(* CODESYS project RepoTestGitCodesys2

Project tree, tasks and I/O mapping:
  Device : CODESYS Control Win V3, 3S - Smart Software Solutions GmbH, version 3.5.19.50
    application Application
      libraries: Standard, 3.5.18.0 (System); Util, 3.5.19.0 (System); Building Automation, 1.0.0.0 (CODESYS Group); CmpBitmapPool, * (System); BASIC, 3.31 (OSCAT); SysTime, 3.5.17.0 (System); SysTypes Interfaces, * (System)
      task AlarmManagerTask (cyclic, interval 50 ms, priority 31) calls AlarmManager.Alarm_Prg
      task MainTask (cyclic, interval t#20ms, priority 1) calls PLC_PRG, test_CFC
      task VISU_TASK (cyclic, interval 100 ms, priority 31) calls VisuElems.Visu_Prg
      Alarm Configuration
        alarm class Alarm (priority 0, acknowledge ACK)
        AlarmStorage
        alarm class Error (priority 10, acknowledge REP)
        alarm class Info (priority 100, acknowledge REP)
        text list List_alarm
        alarm group List_alarm
            0 [Alarm]: Comparison Equal, ExpressionToCompare TRUE, Expression (Reaktor1.Pause.PP00_LT01.WH OR Reaktor1.Innpumping.PP00_LT01.WH) - "Høgt nivå mottakstankl"
            1 [Alarm]: Comparison Equal, ExpressionToCompare TRUE, Expression (Reaktor1.Pause.PP00_LT01.WL OR Reaktor1.Innpumping.PP00_LT01.WL) - "Lavt nivå mottakstank"
            10 [Alarm]: Comparison Equal, ExpressionToCompare TRUE, Expression ((Reaktor2.Pause.PP02_LT02.WL OR Reaktor2.Innpumping.PP02_LT02.WL) OR Reaktor2.Uttaping.PP02_LT02.WL)
            11 [Alarm]: Comparison Equal, ExpressionToCompare TRUE, Expression GVL_Inputs.IA01_PR01_WH
            12 [Alarm]: Comparison Equal, ExpressionToCompare TRUE, Expression GVL_Inputs.IA01_PR01_WL
            13 [Alarm]: Comparison Equal, ExpressionToCompare TRUE, Expression GVL_Inputs.Water_sensor
            2 [Alarm]: Comparison Equal, ExpressionToCompare TRUE, Expression GVL_Inputs.WH_Overflow - "Anlegg i overløp"
            3 [Alarm]: Comparison Equal, ExpressionToCompare TRUE, Expression GVL_Inputs.PA01_PR01_WH
            4 [Alarm]: Comparison Equal, ExpressionToCompare TRUE, Expression GVL_Inputs.PA01_PR01_WL
            5 [Alarm]: Comparison Equal, ExpressionToCompare TRUE, Expression GVL_Inputs.PA02_PR01_WH
            6 [Alarm]: Comparison Equal, ExpressionToCompare TRUE, Expression GVL_Inputs.PA02_PR01_WL
            7 [Alarm]: Comparison Equal, ExpressionToCompare TRUE, Expression ((Reaktor1.Pause.PP01_LT01.WH OR Reaktor1.Innpumping.PP01_LT01.WH) OR Reaktor1.Uttaping.PP01_LT01.WH)
            8 [Alarm]: Comparison Equal, ExpressionToCompare TRUE, Expression ((Reaktor1.Pause.PP01_LT01.WL OR Reaktor1.Innpumping.PP01_LT01.WL) OR Reaktor1.Uttaping.PP01_LT01.WL)
            9 [Alarm]: Comparison Equal, ExpressionToCompare TRUE, Expression ((Reaktor2.Pause.PP02_LT02.WH OR Reaktor2.Innpumping.PP02_LT02.WH) OR Reaktor2.Uttaping.PP02_LT02.WH)
        text list List_Error
        alarm group List_Error
            0 [Error]: Comparison Equal, ExpressionToCompare TRUE, Expression GVL_Inputs.XF_Huber - "Feilsignal grovrist"
            1 [Error]: Comparison Equal, ExpressionToCompare TRUE, Expression Reaktor1.Pause.PP00_LT01.YF OR Reaktor1.Innpumping.PP00_LT01.YF - "Feil på trykkgivar mottakstank"
            10 [Error]: Comparison Equal, ExpressionToCompare TRUE, Expression ((Reaktor1.Innpumping.PP01_PS01.YF = TRUE) AND (Reaktor1.Innpumping.PP01_PS01.YFI = 6)) - "Feil matepumpe 1, safeguard blocking konflikt"
            11 [Error]: Comparison Equal, ExpressionToCompare TRUE, Expression ((Reaktor1.Innpumping.PP01_PS01.YF = TRUE) AND (Reaktor1.Innpumping.PP01_PS01.YFI = 7)) - "Feil matepumpe 1, safeguard mangel tilbakemelding"
            12 [Error]: Comparison Equal, ExpressionToCompare TRUE, Expression ((Reaktor1.Innpumping.PP01_PS01.YF = TRUE) AND (Reaktor1.Innpumping.PP01_PS01.YFI = 8)) - "Feil matepumpe 1, tap av aktivering"
            13 [Error]: Comparison Equal, ExpressionToCompare TRUE, Expression GVL_Inputs.PP01_PS01_XF - "Motorvern matepumpe 1 utløyst"
            14 [Error]: Comparison Equal, ExpressionToCompare TRUE, Expression ((Reaktor1.Innpumping.PP02_PS01.YF = TRUE) AND (Reaktor1.Innpumping.PP02_PS01.YFI = 1)) - "Feil matepumpe 2, mista tilbakemelding høg"
            15 [Error]: Comparison Equal, ExpressionToCompare TRUE, Expression ((Reaktor1.Innpumping.PP02_PS01.YF = TRUE) AND (Reaktor1.Innpumping.PP02_PS01.YFI = 2))
            16 [Error]: Comparison Equal, ExpressionToCompare TRUE, Expression ((Reaktor1.Innpumping.PP02_PS01.YF = TRUE) AND (Reaktor1.Innpumping.PP02_PS01.YFI = 3))
            17 [Error]: Comparison Equal, ExpressionToCompare TRUE, Expression ((Reaktor1.Innpumping.PP02_PS01.YF = TRUE) AND (Reaktor1.Innpumping.PP02_PS01.YFI = 4))
            18 [Error]: Comparison Equal, ExpressionToCompare TRUE, Expression ((Reaktor1.Innpumping.PP02_PS01.YF = TRUE) AND (Reaktor1.Innpumping.PP02_PS01.YFI = 5))
            19 [Error]: Comparison Equal, ExpressionToCompare TRUE, Expression ((Reaktor1.Innpumping.PP02_PS01.YF = TRUE) AND (Reaktor1.Innpumping.PP02_PS01.YFI = 6))
            2 [Error]: Comparison Equal, ExpressionToCompare TRUE, Expression Reaktor1.Pause.PP00_LS01.YF OR Reaktor1.Innpumping.PP00_LS01.YF - "Feil på nivåvippe lav mottakstank"
            20 [Error]: Comparison Equal, ExpressionToCompare TRUE, Expression ((Reaktor1.Innpumping.PP02_PS01.YF = TRUE) AND (Reaktor1.Innpumping.PP02_PS01.YFI = 7))
            21 [Error]: Comparison Equal, ExpressionToCompare TRUE, Expression ((Reaktor1.Innpumping.PP02_PS01.YF = TRUE) AND (Reaktor1.Innpumping.PP02_PS01.YFI = 8))
            22 [Error]: Comparison Equal, ExpressionToCompare TRUE, Expression GVL_Inputs.PP02_PS01_XF
            23 [Error]: Comparison Equal, ExpressionToCompare TRUE, Expression ((Reaktor1.Innpumping.PP01_VP01.YF = TRUE) AND (Reaktor1.Innpumping.PP01_VP01.YF = 1))
            24 [Error]: Comparison Equal, ExpressionToCompare TRUE, Expression ((Reaktor1.Innpumping.PP01_VP01.YF = TRUE) AND (Reaktor1.Innpumping.PP01_VP01.YF = 2))
            25 [Error]: Comparison Equal, ExpressionToCompare TRUE, Expression ((Reaktor1.Innpumping.PP01_VP01.YF = TRUE) AND (Reaktor1.Innpumping.PP01_VP01.YF = 3))
            26 [Error]: Comparison Equal, ExpressionToCompare TRUE, Expression ((Reaktor1.Innpumping.PP01_VP01.YF = TRUE) AND (Reaktor1.Innpumping.PP01_VP01.YF = 4))
            27 [Error]: Comparison Equal, ExpressionToCompare TRUE, Expression ((Reaktor1.Innpumping.PP01_VP01.YF = TRUE) AND (Reaktor1.Innpumping.PP01_VP01.YF = 5))
            28 [Error]: Comparison Equal, ExpressionToCompare TRUE, Expression ((Reaktor1.Innpumping.PP01_VP01.YF = TRUE) AND (Reaktor1.Innpumping.PP01_VP01.YF = 6))
            29 [Error]: Comparison Equal, ExpressionToCompare TRUE, Expression ((Reaktor1.Innpumping.PP01_VP01.YF = TRUE) AND (Reaktor1.Innpumping.PP01_VP01.YF = 7))
            3 [Error]: Comparison Equal, ExpressionToCompare TRUE, Expression (Reaktor1.Pause.PP00_LS02.YF OR Reaktor1.Innpumping.PP00_LS02.YF) - "Feil på nivåvippe høg mottakstank"
            4 [Error]: Comparison Equal, ExpressionToCompare TRUE, Expression GVL_Inputs.XF_Overflow - "Feil på trykkgivar overløp"
            5 [Error]: Comparison Equal, ExpressionToCompare TRUE, Expression ((Reaktor1.Innpumping.PP01_PS01.YF = TRUE) AND (Reaktor1.Innpumping.PP01_PS01.YFI = 1)) - "Feil matepumpe 1, mista tilbakemeldig høg"
            6 [Error]: Comparison Equal, ExpressionToCompare TRUE, Expression ((Reaktor1.Innpumping.PP01_PS01.YF = TRUE) AND (Reaktor1.Innpumping.PP01_PS01.YFI = 2)) - "Feil matepumpe 1, mista tilbakemelding lav"
            7 [Error]: Comparison Equal, ExpressionToCompare TRUE, Expression ((Reaktor1.Innpumping.PP01_PS01.YF = TRUE) AND (Reaktor1.Innpumping.PP01_PS01.YFI = 3)) - "Feil matepumpe 1, mangel tilbakemelding høg"
            8 [Error]: Comparison Equal, ExpressionToCompare TRUE, Expression ((Reaktor1.Innpumping.PP01_PS01.YF = TRUE) AND (Reaktor1.Innpumping.PP01_PS01.YFI = 4)) - "Feil matepumpe 1, mangel tilbakemelding lav"
            9 [Error]: Comparison Equal, ExpressionToCompare TRUE, Expression ((Reaktor1.Innpumping.PP01_PS01.YF = TRUE) AND (Reaktor1.Innpumping.PP01_PS01.YFI = 5)) - "Feil matepumpe 1, ekstern feil"
        alarm group List_Info
        text list List_Info
        alarm group List_Warning
        text list List_Warning
        alarm class Warning (priority 30, acknowledge REP)
      function block BUGS [ST]
      Common_Functions/
        program CommonFunctions [CFC]
        function block Pumphouse [CFC]
      function block fbAnalougeAlarm [ST]
      function block fbDigitalAlarm [ST]
      function block fbInnpumping [ST]
      function block fbPause [ST]
      function block fbSwap [ST]
      function block fbTimer [ST]
      function block fbUtrekningar [ST]
      Function blocks/
        function block Fault_Mapping [ST]
        function block fbBehandlaVatn [ST]
        function block fbCAC [ST]
        function block fbDatabehandling [ST]
        function block fbFeilhandtering [ST]
        function block fbHighload [ST]
        function block fbPumphouse [ST]
        function block fbPumpInterlock [ST]
        function block fbReaksjon [ST]
        function block fbSedementering [ST]
        function block fbSivbedRotation [ST]
        function block fbSlamutak [ST]
        function block fbUttapping [ST]
        function block Output_Mapping [ST]
      Function blocks/
      Functions/
        function Volume_Rectangle [ST]
      Global Variable Lists/
        global variables GVL_Outputs
        global variables GVL_Rest
      global variables GVL
      global variables GVL_Inputs
      global variables GVL_R1
      global variables GVL_R2
      global variables GVL_Sekvenstider
      global variables GVL_TM
      Heile_R1/
        function block R1_Innpumping [CFC]
        function block R1_Pause [CFC]
        function block R1_Reaksjon [CFC]
        function block R1_Sedementering [CFC]
        function block R1_Slam [CFC]
        function block R1_Uttapping [CFC]
        program Reaktor1 [CFC]
      Heile_R2/
        function block R2_Innpumping [CFC]
        function block R2_Innpumping [CFC]
        function block R2_Pause [CFC]
        function block R2_Pause [CFC]
        function block R2_Reaksjon [CFC]
        function block R2_Sedementering [CFC]
        function block R2_Slam [CFC]
        function block R2_Uttapping [CFC]
        program Reaktor2 [CFC]
        program Reaktor2 [CFC]
      function IEC_Time [ST]
      image pool ImagePool
      function block MA [ST]
      function block MB [ST]
      text list MyStates
      program PLC_PRG [ST]
      program POU [ST]
      function block SBE [ST]
      function block SBV [ST]
      function block SBV [ST]
      function block SBV_ReArranged [ST]
      Simulation/
        function block Analog_I [LD]
        function block Analog_O [LD]
        function block fbTankTest [ST]
        function block fbTankVirk [LD]
        function block fbValveSim [ST]
        function block ManualControl [LD]
        global variables Simu
        program Simulering [CFC]
        program Tank [ST]
      visualisation Simulering
      function block SPE [ST]
      visualisation Symbol
      Test_Blocks/
        function block SBV_1 [ST]
        function block test [ST]
        program Reaktor_2 [CFC]
      program test_CFC [CFC]
      function block test [CFC]
      program test_SFC [SFC]: Init_active
      visualisation Testing
      Tilstandsmaskin/
      function block tmReactor1 [ST]
      program Utrekningar [ST]
      function VolumReaktor [ST]
  libraries: VisuSymbols, 4.5.0.0 (System)
  5ce3da45-db07-42e7-a21c-a00fff4ed8f6|C:\Users\Peter\Downloads\GreenBlaser.png
  5ce3da45-db07-42e7-a21c-a00fff4ed8f6|C:\Users\Peter\Downloads\GreenPump90d.png
  5ce3da45-db07-42e7-a21c-a00fff4ed8f6|C:\Users\Peter\Downloads\GreenPump.png
  5ce3da45-db07-42e7-a21c-a00fff4ed8f6|C:\Users\Peter\Downloads\GreenValve-removebg-preview.png
  5ce3da45-db07-42e7-a21c-a00fff4ed8f6|C:\Users\Peter\Downloads\SARA (2).png
  5ce3da45-db07-42e7-a21c-a00fff4ed8f6|C:\Users\Peter\Downloads\WhiteBlaser.png
  5ce3da45-db07-42e7-a21c-a00fff4ed8f6|C:\Users\Peter\Downloads\WhitePump90d.png
  5ce3da45-db07-42e7-a21c-a00fff4ed8f6|C:\Users\Peter\Downloads\WhitePump.png
  5ce3da45-db07-42e7-a21c-a00fff4ed8f6|C:\Users\Peter\Downloads\WhiteValve-removebg-preview.png
  5ce3da45-db07-42e7-a21c-a00fff4ed8f6|C:\Users\Peter\OneDrive - Høgskulen på Vestlandet\Mango_Disk\Bachelor RA200 Sande\Dokumentasjon\P&ID\Eldre versjoner\SARA_P&ID_rev2.drawio.png
  5ce3da45-db07-42e7-a21c-a00fff4ed8f6|C:\Users\Peter\OneDrive - Høgskulen på Vestlandet\Mango_Disk\Bachelor RA200 Sande\Dokumentasjon\P&ID\P&ID Automatisk styrt.png
  5ce3da45-db07-42e7-a21c-a00fff4ed8f6|C:\Users\Peter\OneDrive - Renasys\Dokumenter\GreenValve90d.png
  5ce3da45-db07-42e7-a21c-a00fff4ed8f6|C:\Users\Peter\OneDrive - Renasys\Dokumenter\WhiteValve90d.png
  5ce3da45-db07-42e7-a21c-a00fff4ed8f6|C:\Users\Peter\OneDrive - Renasys\Skrivebord\GreenValve.png
  5ce3da45-db07-42e7-a21c-a00fff4ed8f6|C:\Users\Peter\OneDrive - Renasys\Skrivebord\WhiteValve.png
  5ce3da45-db07-42e7-a21c-a00fff4ed8f6|C:\Users\Peter\OneDrive\Skrivebord\test.png
  GlobalImagePool
  text list GlobalTextList
*)

// Device/Application/GVL
{attribute 'qualified_only'}


VAR_GLOBAL
	lvlTransmitter_Mottak : REAL;
	
END_VAR

// Device/Application/GVL_Inputs
{attribute 'qualified_only'}
VAR_GLOBAL
	
END_VAR

// Device/Application/GVL_R1
{attribute 'qualified_only'}
VAR_GLOBAL
	// Reaktor 1 INPUT	
	SekvensPauseOK					: BOOL;		// Sekvense Pause 			gjennomført
	SekvensInnpumpingOK				: BOOL;		// Sekvense Innpumping  	gjennomført
	SekvensReaksjonOK				: BOOL;		// Sekvense Reaksjon 		gjennomført
	SekvensSedimenteringOK			: BOOL;		// Sekvense Sedimentering 	gjennomført
	SekvensUttappingOK				: BOOL;		// Sekvense Uttapping 		gjennomført

	// Reaktor 1 OUTPUT
	Pause							: BOOL;		// [TRUE] Aktiv Sekvens Pause
	Innpumping 						: BOOL;		// [TRUE] Aktiv Sekvens Innpumping
	Reaksjon 						: BOOL;		// [TRUE] Aktiv Sekvens Reaksjon
	Sedimentering 					: BOOL;		// [TRUE] Aktiv Sekvens Sedimentering
	Uttapping						: BOOL;		// [TRUE] Aktiv Sekvens Uttapping
	
	// Reaktor 1 Sekvens Tider	
	SekvenstidInnpumping			: TIME;		// Maks tid innpumpingssekvens
	SekvenstidReaksjon				: TIME;		// Maks tid reaksjonssekvens
	SekvenstidSedimentering			: TIME;		// Maks tid sedimenteringssekvens
	SekvenstidUttapping  			: TIME;		// Maks tid Uttapping
	
	// Reaktor 1 Reaksjonstider
	GangtidAnoks					: TIME;		// Gangtid Anoks reaksjonsfase 
	GangtidAerob					: TIME;		// Gangtid Aerob reaksjonsfase
	GangtidKjemikalieDosering		: TIME;		// Gangtid Kjemikaliepumpe
	SikkerheitsIntervallKjemikalie	: TIME;		// Tid mellom ferdig kjemikaliedosering og slutt reaksjonsfase : SekvenstidReaksjon - (GangtidKjemikalieDosering + SikkerheitsIntervallKjemikalie)
END_VAR

// Device/Application/GVL_R2
{attribute 'qualified_only'}
VAR_GLOBAL
	// Reaktor 2 INPUT	
	SekvensPauseOK					: BOOL;		// Sekvense Pause 			gjennomført
	SekvensInnpumpingOK				: BOOL;		// Sekvense Innpumping  	gjennomført
	SekvensReaksjonOK				: BOOL;		// Sekvense Reaksjon 		gjennomført
	SekvensSedimenteringOK			: BOOL;		// Sekvense Sedimentering 	gjennomført
	SekvensUttappingOK				: BOOL;		// Sekvense Uttapping 		gjennomført

	// Reaktor 2 OUTPUT
	Pause							: BOOL;		// [TRUE] Aktiv Sekvens Pause							
	Innpumping 						: BOOL;		// [TRUE] Aktiv Sekvens Innpumping
	Reaksjon 						: BOOL;		// [TRUE] Aktiv Sekvens Reaksjon
	Sedementering 					: BOOL;		// [TRUE] Aktiv Sekvens Sedimentering
	Uttapping						: BOOL;		// [TRUE] Aktiv Sekvens Uttapping
	
	// Reaktor 2 Sekvens Tider
	SekvenstidInnpumping			: TIME;		// Maks tid innpumpingssekvens
	SekvenstidReaksjon				: TIME;		// Maks tid reaksjonssekvens
	SekvenstidSedimentering			: TIME;		// Maks tid sedimenteringssekvens
	SekvenstidUttapping  			: TIME;		// Maks tid Uttapping
	
	// Reaktor 2 Reaksjonstider
	GangtidAnoks					: TIME;		// Gangtid Anoks reaksjonsfase
	GangtidAerob					: TIME;		// Gangtid Aerob reaksjonsfase
	GangtidKjemikalie				: TIME;		// Gangtid Kjemikaliepumpe
	SikkerheitsIntervallKjemikalie	: TIME;		// Tid mellom ferdig kjemikaliedosering og slutt reaksjonsfase : SekvenstidReaksjon - (GangtidKjemikalieDosering + SikkerheitsIntervallKjemikalie)
END_VAR

// Device/Application/GVL_Sekvenstider
{attribute 'qualified_only'}
VAR_GLOBAL	
	TidInnpumpingMaks			: TIME := T#10S;
	TidReaksjon					: TIME := T#3S;
	TidSedimentering			: TIME := T#3S;
	TidUttapping  				: TIME := T#3S;
END_VAR

// Device/Application/GVL_TM
{attribute 'qualified_only'}
VAR_GLOBAL
	
	// Reaktor 1
	Pause1						: BOOL;							//
	Innpumping1 				: BOOL;
	Innpumping_Pause1			: BOOL;
	Reaksjon1 					: BOOL;
	Sedementering1 				: BOOL;
	Uttapping1					: BOOL;
	
	// Reaktor 2
	Pause2						: BOOL;							//
	Innpumping2 				: BOOL;
	Innpumping_Pause2			: BOOL;
	Reaksjon2 					: BOOL;
	Sedementering2 				: BOOL;
	Uttapping2					: BOOL;
	
	// Til tilstandsmaskin
	PauseReaktor1OK				: BOOL;
	
	InnpumpingReaktor1OK		: BOOL; 
	InnpumpingReaktor1Pause		: BOOL;
END_VAR

// Device/Application/Global Variable Lists/GVL_Outputs
{attribute 'qualified_only'}
VAR_GLOBAL
END_VAR

// Device/Application/Global Variable Lists/GVL_Rest
{attribute 'qualified_only'}
VAR_GLOBAL
	
	MottakstankNivaa	: REAL;
	MottakstankVolum	: REAL;
	siSivState			: INT;
	GangerPrSivBed		: INT;

END_VAR

// Device/Application/Simulation/Simu
{attribute 'qualified_only'}
VAR_GLOBAL
	XE	: BOOL := TRUE;
	LA	: BOOL;
	
	MTankNivaa		: REAL;
	R1Nivaa			: REAL;
	FlowInlet		: INT;
	FlowOutletR1	: INT;
	
	PP01_VP01_YF 	: BOOL;
	PP02_VP01_YF 	: BOOL;
	TW02_VH01_YF 	: BOOL;
	
	PP01_PS01_YF 	: BOOL;
	PP02_PS01_YF 	: BOOL;
	PA01_BL01_YF 	: BOOL;
	CH00_PH01_YF 	: BOOL;
END_VAR

// Device/Application/PLC_PRG
PROGRAM PLC_PRG
VAR

LS_LOW   : MB;
LS_HIGH  : MB;
PT_Tank	 : MA;
PT_R1	 : MA;
PT_R2	 : MA;
M1		 : SPE;
M2		 : SPE;
Valve1   : SBV;
Valve2	 : SBV;
Swap	 : fbSwap;

END_VAR

//Test();

LS_LOW();
LS_HIGH();
PT_TANK();
M1();
M2();
Valve1();
Valve2();
test();

// Beginning of the code :

IF LS_LOW.X THEN
	
	// Retracting Low Commands
	M1.XL		:= FALSE;
	Valve1.XL	:= FALSE;

	// Sending High Commands
	M1.XH 		:= TRUE;
	Valve1.XH 	:= TRUE;
	
ELSIF (NOT LS_LOW.X) THEN
	
	// Retracting HIGH Commands
	M1.XH		:= FALSE;
	Valve1.XH	:= FALSE;

	// Sending LOW Commands
	M1.XL 		:= TRUE;
	Valve1.XL 	:= TRUE;
	
END_IF

END_PROGRAM

// Device/Application/Test_Blocks/test
FUNCTION_BLOCK test
VAR_INPUT
END_VAR
VAR_OUTPUT
END_VAR
VAR
END_VAR

END_FUNCTION_BLOCK

// Device/Application/test
FUNCTION_BLOCK test
VAR_INPUT
	XE						: BOOL;			// Input from state machine
END_VAR
VAR_OUTPUT
	Y						: BOOL;			// Output to state machine
END_VAR

VAR
	// INPUT BLOCKS
	PP00_LS02   			: MB;			// Mottasktank vippe lav, call "Monitor Binary" 
	PP00_LS01  				: MB;			// Mottasktank vippe høg, call "Monitor Binary" 
	PP00_LT01	 			: MA;			// Mottasktank nivåmålar, call "Monitor Analog"
	PP01_LT01	 			: MA;			// Reaktor 1 nivåmålar,   call "Monitor Analog"
	
	// OUTPUT BLOCKS
	PA01_BL01				: SBE;			// Reaktor 1 blåser,	 call "Switch Binary Electrical"
	PP01_PS01		 		: SBE;			// Matepumpe 1,			 call "Switch Binary Electrical"
	PP02_PS01		 		: SBE;			// Matepumpe 2,			 call "Switch Binary Electrical"
	PP01_VP01   			: SBV;			// Reaktor 1 inn ventil, call "Switch Binary Valve"
	
	// FUNCTION BLOCKS
	Sekvens_Innpumping		: fbInnpumping;	// Innpumping logic,         call "fbInnpumping"
	Sim						: fbValveSim;	// Feedback balve simulator, call "fbValveSim"
END_VAR

VAR_TEMP		
	// FUNCTION CONTROL PARAMETERS
	PYHR				: REAL := 100;		// (Mottasktank nivåmålar & Reaktor 1 nivåmålar) MA Parameter Y high range
	PYLR				: REAL := 0;		// (Mottasktank nivåmålar & Reaktor 1 nivåmålar) MA Parameter Y low range
	PP00_LT01_PAHH		: REAL := 32;		// (Mottasktank nivåmålar) 						 MA Parameter high high action
	PP00_LT01_PALL		: REAL := 5;		// (Mottasktank nivåmålar) 						 MA Parameter low low action
	PP01_LT01_PAHH		: REAL := 90;		// (Reaktor 1 nivåmålar)   						 MA Parameter low low action 
	END_VAR

// -------------------------------------------------------------------------------------------------------------------------------------------------IN BLOCKS----------------------------------------------------------------------------------------------------------------------------------------------------------------------------------------------------------
// Mottakstank vippe høg
// INPUTS
// OUTPUTS
PP00_LS01(X := GVL_Inputs.PP00_LS01_X); // MB
// Mottakstank vippe lav
// INPUTS
// OUTPUTS
PP00_LS02(X := GVL_Inputs.PP00_LS02_X); // MB
// Mottakstank Nivåmåling
// INPUTS
PP00_LT01(
    X := GVL_Inputs.PP00_LT01_X,
    PAHH := PP00_LT01_PAHH,
    PALL := PP00_LT01_PALL,
    PYHR := PYHR,
    PYLR := PYLR); // MA
// OUTPUTS
GVL_Rest.MottakstankNivaa := PP00_LT01.Y;
// Reaktor 1 Nivåmåling
// INPUTS
PP01_LT01(X := GVL_Inputs.PP01_LT01_X, PAHH := PP01_LT01_PAHH, PYHR := PYHR, PYLR := PYLR); // MA
// OUTPUTS
GVL_R1.Nivaa := PP01_LT01.Y;
// ------------------------------------------------------------------------------------------------------------------------------------------------- CODE ----------------------------------------------------------------------------------------------------------------------------------------------------------------------------------------------------------
Sekvens_Innpumping(
    AHH_SendingTank := PP00_LT01.AHH,
    ALL_SendingTank := PP00_LT01.ALL,
    HH_SendingTank := PP00_LS01.Y,
    LL_Sending_Tank := PP00_LS02.Y,
    AHH_ReceivingTank := PP01_LT01.AHH,
    ALL_ReceivingTank := PP01_LT01.ALL,
    XGH_RValve := PP01_VP01.BCH,
    XGL_RValve := PP01_VP01.BCL,
    XGL_Pump1 := PP01_PS01.BCL,
    XGL_Pump2 := PP02_PS01.BCL,
    XE := XE,
    PIT := GVL_R1.SekvenstidInnpumping,
    PTI := GVL_R1.IntervallBlaser,
    PTD := GVL_R1.GangtidBlaser); // fbInnpumping
// Reaktor 1 blåser
// INPUTS
PA01_BL01(
    XGH := PA01_BL01.Y,
    XH := Sekvens_Innpumping.YH_Blower,
    XL := Sekvens_Innpumping.YL_Blower,
    XE := GVL_R1.Innpumping,
    LA := Simu.LA); // SBE
GVL_R1.Innpumping_PA01_BL01_YF := PA01_BL01.YF;
Y := Sekvens_Innpumping.Y;
// ------------------------------------------------------------------------------------------------------------------------------------------------- OUT BLOCKS  ---------------------------------------------------------------------------------------------------------------------------------------------------------------------------------------------------
// Inntaktspumpe 1
// INPUTS
PP01_PS01(
    XGH := PP01_PS01.Y,
    XH := Sekvens_Innpumping.YH_Pump1,
    XL := Sekvens_Innpumping.YL_Pump1,
    XE := GVL_R1.Innpumping,
    LA := Simu.LA); // SBE
GVL_R1.PP01_PS01_YF := PP01_PS01.YF;
// OUTPUTS
GVL_R1.PP01_PS01_Y := PP01_PS01.Y;
// Inntaktspumpe 2
// INPUTS
PP02_PS01(
    XGH := PP02_PS01.Y,
    XH := Sekvens_Innpumping.YH_Pump2,
    XL := Sekvens_Innpumping.YL_Pump2,
    XE := GVL_R1.Innpumping,
    LA := Simu.LA); // SBE
// OUTPUTS
GVL_R1.PP02_PS01_Y := PP02_PS01.Y;
GVL_R1.PP02_PS01_YF := PP02_PS01.YF;
// OUTPUTS
GVL_R1.Innpumping_PA01_BL01 := PA01_BL01.Y;
// Reaktor 1 inn ventil
// INPUTS
PP01_VP01(
    XGH := PP01_VP01.BCH,
    XGL := PP01_VP01.BCL,
    XH := Sekvens_Innpumping.YH_RValve,
    XL := Sekvens_Innpumping.YL_RValve,
    LA := Simu.LA); // SBV
// OUTPUTS
GVL_Outputs.PP01_VP01_Y := PP01_VP01.Y;
GVL_R1.PP01_VP01_YF := PP01_VP01.YF;
GVL_R1.PP01_VP01_BCH := PP01_VP01.BCH;

END_FUNCTION_BLOCK

// Device/Application/SBE
FUNCTION_BLOCK SBE
//The SBE function template shall be used for binary (on/off) control of flow element of medium 
//(electricity, heat or fluid). The controlled element is a unit, e.g. motor, pump, heater, fan etc.

VAR_INPUT
	{Signal FROM MCC, running status high (XGH = 1 is motor 
running)}
	XGH 		: BOOL; // Pos high feedback (MCC)	
	{XH = 1 (positive edge) set Y TO 1 in auto mode.)}
	XH 			: BOOL; // External set high 
	{XL = 1 (positive edge) set Y TO 0 in auto mode. XL is 
dominant over XH.}
	XL			: BOOL; // External set low
	{XOH = 1 set Y TO 1 in outside mode.}
	XOH 		: BOOL; // External outside set high
	{XOL = 1 set Y TO 0 in outside mode.}
	XOL			: BOOL; //External outside set low
	{Loop failure, e.g. I/O card broken}
	XF			: BOOL; // External fault
	{XE = 1 is required FOR a start. The effect on Y when XE goes 
low while running will be defined by parameter.}
	XE			: BOOL; // External enabled (MCC)
	{Safeguarding – LSH = 1. Overrule operator possibility TO 
operate Start/Stop and Auto/Manual. Locks template in 
manual mode and Y to 1 regardless of failure state. Input is 
subject to blocking. When signal goes low, the template 
remains in manual mode and Y = 1}
	LSH			: BOOL; // Lock safeguarding high
	{Safeguarding – LSL = 1 Overrule operator possibility TO 
operate Start/Stop and Auto/Manual. Locks template to 
manual mode and Y to 0 regardless of failure state. Input is 
subject to blocking. When signal goes low, the template 
remains in manual mode and Y = 0}
	LSL			: BOOL; // Lock safeguarding low
	{Safeguarding – FSH = 1 Overrule operator possibility TO 
operate Start/Stop. Sets Y to1 regardless of failure state. 
When signal is reset, the template will react to actual 
terminal statuses again. Signal is subject to blocking. If in 
Manual mode, the output (Y) remains 1 after signal returns 
to normal. }
	FSH			: BOOL; // Force safeguarding high
	{Safeguarding FSH = 0 Overrule operator possibility TO 
operate Start/Stop. Sets to 0 regardless of failure state. 
When signal is reset, the template will react to actual 
terminal statuses again. Signal is subject to blocking.
If in manual mode, the output (Y) remains 0 after signal 
returns to normal.}
	FSL			: BOOL; // Force safeguarding low
	{Permissive TO start when FDH = 0 AND prevents equipment 
from being started when FDH = 1.
Signal is subject to blocking.}
	FDH			: BOOL; // Force disable transition high
	{Permissive TO stop when FDL = 0 AND prevents equipment FROM being stopped when FDL = 1.
Signal is subject to blocking.}
	FDL 		: BOOL;	// Force transition low
	{FB = 1. Safeguarding ACTION LSH, LSL, FSH, FSL AND FDH AND FDL will be blocked}
	FB			: BOOL;	// Force blocking
	{FU = 1. Alarm annunciation is suppressed, YF = 0. AND statuses XF, XE AND XGH are neglected. }
	FU			: BOOL;	// Force supression
	{Locks the template in auto mode. When LA is reset, the template remains in auto mode.}
	LA			: BOOL; // Lock auto
	{Locks the template in manual mode. When LM is reset, the template remains in manual mode}
	LM			: BOOL;	// Lock manual
	{Locks the template in outside mode. When LO goes low the template will be set TO manual mode. }
	LO			: BOOL; // Lock outside
END_VAR
VAR_OUTPUT
	{Command TO flow element. Start Y = 1 AND stop Y = 0.}
	Y		: BOOL; // Normal function output
	{Pulse start command YH = 1 (one pulse)}
	YH		: BOOL; // Pulsed normal function output high
	{Pulse stop command YL = 1 (one pulse).}
	YL		: BOOL;	// Pulsed normal function output low
	{Set YF = 1 IF XF = 1 OR feedback TIME exceeded OR change in feedback WHILE in run OR stop OR XE = 0}
	YF		: BOOL; // Function failed
	{Output Y compared TO feedback position high LIMIT switch AND validated as TRUE (set BCH = 1 IF Y = 1 AND XGH = 1). XF has no impact on BCH}
	BCH		: BOOL; // Output position high confirmed
	{Output Y compared TO feedback position low LIMIT switch AND validated as TRUE (set BCL = 1 IF Y = 0 AND XGH = 0). XF has no impact on BCL.}
	BCL		: BOOL; // Output position low confirmed
	{BS = 1 IF ANY safeguarding input is active.}
	BS		: BOOL; // Status safeguarding
	{BB = 1 when block FROM operator station is TRUE OR FB = 1}
	BB		: BOOL; // Status blocked 
	{BU = 1 when suppressed FROM operator station is TRUE OR FU = 1}
	BU		: BOOL; // Status supressed
	{BA = 1 when in auto mode.}
	BA		: BOOL; // Status auto/man
	{BO = 1 when outside mode set FROM operator station OR LO = 1}
	BO		: BOOL; // Status outside
	{BXH = 1 when SBE is in auto AND XH = 1 OR start signal FROM SBC.}
	BXH		: BOOL; // Status external set high
	{BXL = 1 when SBE is in auto AND XL = 1 OR stop signal FROM 
SBC.}
	BXL		: BOOL; // Status external set low
	
END_VAR
VAR
END_VAR

//Mangler

END_FUNCTION_BLOCK

// Device/Application/fbInnpumping
FUNCTION_BLOCK fbInnpumping

VAR_INPUT
	Sending_Tank_AHH					: BOOL;					// Mottaktstank nivåmåler
	Sending_Tank_ALL					: BOOL;					// Mottaktstank nivåmåler
	Sending_Tank_LS_High				: BOOL;					// Inngang for vippe i mottakstank HIGH HIGH
	Sending_Tank_LS_Low					: BOOL;					// Inngang for vippe i mottakstank LOW LOW 
	
	Reciving_Tank_AHH					: BOOL;					// Reaktor AHH nivå¨måler
	Reciving_Tank_ALL					: BOOL;					// Reaktor ALL nivå måler
	
	Valve_Confirmed_Open				: BOOL;
	Valve_Confirmed_Close				: BOOL;
	Pump1_Confirmed_Stopped				: BOOL;
	Pump2_Confirmed_Stopped				: BOOL;
END_VAR


VAR_OUTPUT
	Valve_Open							: BOOL;
	Valve_Close							: BOOL;
	
	Pump_1_Start						: BOOL;
	Pump_1_Stopp						: BOOL;
	Pump_2_Start						: BOOL;
	Pump_2_Stopp						: BOOL;
END_VAR

VAR
	
	PumpSwitch					: fbSwap;

	InnpumpingTimer				: fbTimer;

//END_VAR

//VAR_TEMP	
	tbSending_Tank_AHH						: BOOL;						// ER Høg om nivå er over tillatt innpumping
	tbSending_Tank_ALL						: BOOL;						// ER Høg om nivå er over tillatt innpumping
	tbSending_Tank_LS_High					: BOOL;
	tbSending_Tank_LS_Low					: BOOL;
	tbReciving_Tank_AHH						: BOOL;
	
	tbPump									: BOOL;
END_VAR

VAR CONSTANT

END_VAR


// Populate temporaries
tbSending_Tank_AHH								:= Sending_Tank_AHH;
tbSending_Tank_ALL								:= Sending_Tank_ALL;
tbSending_Tank_LS_High							:= Sending_Tank_LS_High;
tbSending_Tank_LS_Low							:= Sending_Tank_LS_Low;	
tbReciving_Tank_AHH								:= Reciving_Tank_AHH;

// Populate and start timers
//InnpumpingTimer();
//InnpumpingTimer.PTDH					:= GVL_Sekvenstider.TidInnpumpingMaks;


// NB! Dersom reaktoren ikkje klarer og tømme seg, foreksempel visst uttappingrøyret går tett vil tilstandsmaskina hoppe rett forbi innpumpingsfasen og gå rett ifrå pause til reaksjon.



IF GVL_TM.Innpumping1 THEN
	
	// pump is started because the water in sending tank is high enough
	IF (tbSending_Tank_AHH OR Sending_Tank_LS_High) THEN // Sjekka betingelser for å gå
		
		//InnpumpingTimer.X					:= TRUE;	// start timer
		
		// Opne ventil tilhøyrande
		Valve_Close			:= FALSE;
		Valve_Open 			:= TRUE;
				
		// Velge & Starte Pumpe		
		PumpSwitch.X 		:= TRUE;
		
		// Saving a bool memory based on wich output from Switch that comes back true
		IF (PumpSwitch.Y1) THEN
			tbPump			:= TRUE;
		ELSIF (PumpSwitch.Y2) THEN
			tbPump			:= FALSE;
		END_IF

		// Starts pump based on saved memory
		IF (tbPump AND Valve_Confirmed_Open) THEN
			Pump_1_Stopp	:= FALSE;
			Pump_1_Start	:= TRUE;
		ELSIF (NOT tbPump AND Valve_Confirmed_Open) THEN
			Pump_2_Stopp	:= FALSE;
			Pump_2_Start	:= TRUE;
		END_IF
		
	END_IF
	

	// If pumping is stopped because of low water in sending tank.	
	IF (Sending_Tank_ALL OR Sending_Tank_LS_LOW) THEN
				
		// Stopping running pumps
		IF (tbPump) THEN
			Pump_1_Start	:= FALSE;
			Pump_1_Stopp	:= TRUE;
		ELSIF NOT (tbPump) THEN
			Pump_2_Start	:= FALSE;
			Pump_2_Stopp	:= TRUE;
		END_IF
		
		// Close valve with pump 1 feedback
		IF (tbPump AND Pump1_Confirmed_Stopped) THEN
			Valve_Open	:= FALSE;
			Valve_Close := TRUE;		
		END_IF
		
		// Close valve with pump 2 feedback		
		IF (NOT tbPump AND Pump2_Confirmed_Stopped) THEN
			Valve_Open	:= FALSE;
			Valve_Close := TRUE;		
		END_IF
	END_IF

	// IF pumping is stopped because reciving tank is full or a max time intervall is reached
	IF (Reciving_Tank_AHH ) THEN	 // Sjekka betingelser for å gå vidare til reaksjon // OR InnpumpingTimer.Y 
		
		// Stopping running pumps
		IF (tbPump) THEN
			Pump_1_Start	:= FALSE;
			Pump_1_Stopp	:= TRUE;
		ELSIF NOT (tbPump) THEN
			Pump_2_Start	:= FALSE;
			Pump_2_Stopp	:= TRUE;
		END_IF
				
		// Close valve with pump 1 feedback
		IF (tbPump AND Pump1_Confirmed_Stopped) THEN
			Valve_Open	:= FALSE;
			Valve_Close := TRUE;		
		END_IF
		
		// Close valve with pump 2 feedback		
		IF (NOT tbPump AND Pump2_Confirmed_Stopped) THEN
			Valve_Open	:= FALSE;
			Valve_Close := TRUE;		
		END_IF
		
		// Sending Tilstandmaskin to next state if valve is confirmed closed
		
		IF Valve_Confirmed_Close THEN
			GVL_TM.InnpumpingReaktor1OK := TRUE;
		ELSE
			GVL_TM.InnpumpingReaktor1OK := FALSE;
		END_IF
		
							
	END_IF
END_IF

END_FUNCTION_BLOCK

// Device/Application/Simulation/Tank
PROGRAM Tank
VAR
	Kall	: fbTankVirk;
END_VAR

Kall(PumpPower := Simu.PumpFlowLS, IdleTime := Simu.IdleTime, FillLevel := Simu.FillLevelLS);

END_PROGRAM

// Device/Application/Simulation/fbTankVirk
FUNCTION_BLOCK fbTankVirk
VAR_INPUT
	PumpPower	: REAL;
	IdleTime	: INT;
END_VAR
VAR_IN_OUT
	FillLevel	: REAL;
END_VAR
VAR
	PumpOutputReal 		: REAL;
	PumpMemory			: ARRAY[0..9999] OF REAL;
	i					: INT;
	PumpMemoryResult	: REAL;
END_VAR

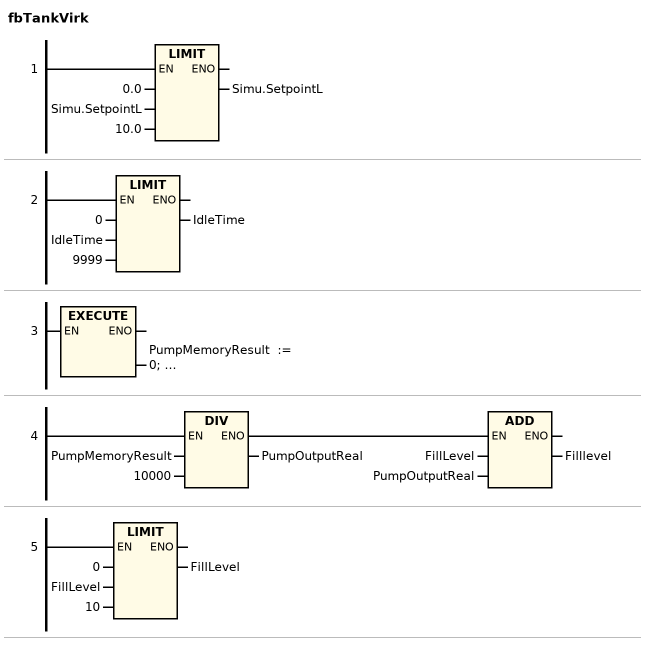
// NETWORK 1
Simu.SetpointL := LIMIT(0.0, Simu.SetpointL, 10.0);

// NETWORK 2
IdleTime := LIMIT(0, IdleTime, 9999);

// NETWORK 3
PumpMemoryResult  := 0;

FOR i := 1 TO IdleTime DO
	PumpMemory[i - 1] := PumpMemory[i];
	PumpMemoryResult := PumpMemoryResult + PumpMemory[i - 1];
END_FOR

PumpMemory[IdleTime] := PumpPower;
PumpMemoryResult := PumpMemoryResult + PumpMemory[IdleTime];
PumpMemoryResult := PumpMemoryResult / IdleTime;

IF Simu.EmptyTank THEN
	FOR i := 1 TO IdleTime DO
		PumpMemory[i] := 0;
	END_FOR
END_IF

// NETWORK 4
PumpOutputReal := PumpMemoryResult / 10000;
Filllevel := FillLevel + PumpOutputReal;

// NETWORK 5
FillLevel := LIMIT(0, FillLevel, 10);

END_FUNCTION_BLOCK

// Device/Application/fbSwap
FUNCTION_BLOCK fbSwap
VAR_INPUT
	X				: BOOL;			// eXternal input
	XF				: BOOL;			// eXternal fault
END_VAR

VAR_OUTPUT
	Y1				: BOOL;			// Output 1
	Y2				: BOOL;			// Output 2
	YF				: BOOL;			// Fault
END_VAR

VAR	
	sbX				: BOOL;			// Static memory eXternal input
	siSwapCase		: SINT;			// Static int Case
END_VAR

VAR_TEMP
	tbX				: BOOL;			// temp eXternal input
	tbY1			: BOOL;			// temp output 1
	tbY2			: BOOL;			// temp output 2
	tbXF			: BOOL;			// temp eXternal fault
	tbYF			: BOOL;			// temp fault
END_VAR

VAR CONSTANT
	ciOutput1		: SINT := 1;	// constant case output 1
	ciOutput2		: SINT := 2;	// constant case output 2
END_VAR

// Populate temoraries
tbX		:= X;
tbXF	:= XF;

// Counter increases by 1 each time X goes high
IF tbX AND NOT sbX THEN
	siSwapCase := siSwapCase + 1;
END_IF

// Retrigger posetive edge
sbx		:= tbx;

// Handles if case is outside limits
IF (siSwapCase > ciOutput2) THEN
	siSwapCase := ciOutput1;
END_IF


// Input and Case
IF tbX THEN	
	CASE siSwapCase OF
		
		ciOutput1: // Statement section case 1 (Only Output Y1)		
			tbY2 := FALSE;
			tbY1 := TRUE;
				
		ciOutput2: // Statement section case 2 (Only Output Y2)
	
			tbY2 := TRUE;
			tbY1 := FALSE;	
	END_CASE
END_IF

IF (tbXF OR (Y1 = TRUE AND Y2 = TRUE)) THEN
	tbYF := TRUE;
ELSE
	tbYF := FALSE;
END_IF

// Writing to outputs
Y1		:= tbY1;
Y2		:= tbY2;
YF		:= tbYF;

END_FUNCTION_BLOCK

// Device/Application/fbTimer

FUNCTION_BLOCK fbTimer
VAR_INPUT
	X 		       : BOOL;			// Input	
	PTDH	       : TIME;			// High Delay
	PTDL		   : TIME;			// Low Delay	
	
	
END_VAR

VAR_OUTPUT
	Y  				: BOOL;			// Limit violation
END_VAR

VAR
	stTimeOn 		: TIME;
	stTimeOff 		: TIME;
	sbDelayBlock    : BOOL;			//Beskyttelse
END_VAR

VAR_TEMP
	ttNow 	: TIME;
	ttTimeOn 	: TIME;
	ttTimeOff 	: TIME;
END_VAR

// Timerblokk designed by MangoIPA Team and is 
// approved by drinkers all around the world



// ttNow gets PLC time
ttNow 								:= TIME();							

// ttTime teller tida
ttTimeON 							:= ttNow - stTimeOn;
ttTimeOff 							:= ttNow - stTimeOff;

// OnDelay
IF X THEN
	sbDelayBlock 					:= FALSE;
	IF(ttTimeOn >= PTDH) THEN
		Y 							:= TRUE;		
	END_IF;
ELSE	
	sbDelayBlock 					:= TRUE;
	stTimeOn  						:= ttNow;
END_IF;

// OffDelay
IF NOT X AND sbDelayBlock THEN
	
	IF(ttTimeOff >= PTDL) THEN
		Y 							:= FALSE;
	END_IF;
ELSE
	stTimeOff  						:= ttNow;	
END_IF;

END_FUNCTION_BLOCK

// Device/Application/MB
FUNCTION_BLOCK MB
VAR_INPUT
	
	X		: BOOL;   					// Normal function input
	XF		: BOOL;  					// External Fault
	RX		: BOOL;  					// Reset latched output
	FB		: BOOL;  					// Force blocking
	FU		: BOOL;  					// Force suppression
	
END_VAR

VAR_INPUT RETAIN
	
	PI		: BOOL 		:= FALSE; 		// Parameter invert input
	PL		: BOOL 		:= FALSE; 		// Parameter latched output
	PT_delay: TIME 		:= T#0S; 		// Parameter time telay alarm
	
END_VAR

VAR_OUTPUT
	
	Y		: BOOL;  					// Normal function output
	YF		: BOOL; 					// Function failed
	BB		: BOOL; 					// Status blocked
	BU		: BOOL; 					// Status suppressed
	BX		: BOOL; 					// Status function input
	
END_VAR

VAR
	
	OS_FB	: BOOL; 					// Operator station blocking on/off
	OS_FU	: BOOL; 					// Operator station suppression on/off
	OS_RX	: BOOL; 					// Reset Latched output	

	sbX 	: BOOL; 					// Posetive edge memory	
	
	fbTimer : fbtimer; 					// Timer FB
	
	
	OS_BB 	: BOOL; 					// Operator staton output (blocked)	
	OS_BU 	: BOOL; 					// Operator station output (Supressed)	
	OS_YF 	: BOOL; 					// Operator station (Alarms)
END_VAR

VAR_TEMP

	tbX		: BOOL;						// Temp normal function input
	tbXF	: BOOL;						// Temp external fault
	tbRX	: BOOL;						// Temp reset latched output
	tbFB	: BOOL;						// Temp force blocking
	tbFU	: BOOL;						// Temp force supression
	
	tbY		: BOOL;						// Temp normal function output
	tbYF	: BOOL;						// Temp function failed
	tbBB	: BOOL;						// Temp status blocked
	tbBU	: BOOL;						// Temp status supressed
	tbBX	: BOOL;						// Temp function input
	
	internal_error: BOOL;				// Temp internal function error
END_VAR


// Populate/Initialize temporaries
tbx 					:= X;
tbXF 					:= XF;
tbRX 					:= RX;
tbFB 					:= FB;
tbFU 					:= FU;

fbTimer.PTDH 			:= PT_delay;
fbtimer();


// FROM OS (Added if functonality is wanted in operating station)
// OS_XB :=
// OS_FU :=
// OS_RX :=

// Handle parameter inverted
IF PI THEN
    tbx 				:= NOT tbx;
END_IF;

// Mode Not latched
IF NOT PL THEN
	fbTimer.X			:=tbX;
END_IF;	
	
// Mode latched
IF PL AND NOT PI THEN	
    // Posetiv edge on X
    IF tbX AND NOT sbX THEN		
		fbTimer.X		:= TRUE;			
    END_IF;

    IF (tbRX OR OS_RX) AND NOT tbX THEN		// Reset
		fbTimer.X 		:= FALSE;
    END_IF;

    // Reset posetiv edge
    sbx 				:= tbX;
END_IF;
    

//Mode latched and inverted
IF PL  AND PI THEN
	
    // Negativ flank detection
    IF tbX AND sbX THEN		
		fbTimer.X		:= TRUE;			
    END_IF;

    IF (tbRX OR OS_RX) AND NOT tbX THEN		//Reset
		fbTimer.X 		:= FALSE;
    END_IF;

    // Reset negative edge
    sbx					:= NOT tbX;
END_IF;
	

// BX always equal to Input
tbBX 					:= tbX;

//Handle timer output
tbY 					:= fbTimer.Y;
 
// Handle Force Supression
IF tbFU OR OS_FU THEN
	
	tbBU 			:= TRUE;
	tbY				:= FALSE;
	tbYF 			:= FALSE;
	
    ELSE
        tbBU 			:= FALSE;
    END_IF;

    // Handle Force block
    IF tbFB OR OS_FB THEN
        tbBB 			:= TRUE;
        tbY 			:= FALSE;
	ELSE
		tbBB 			:= FALSE;
    END_IF;

    // Handle Fault
    IF (tbXF OR internal_error) AND NOT (tbFU) AND NOT (OS_FU) THEN
        tbYF			:= TRUE;
    ELSE
        tbYF 			:= FALSE;
END_IF;


// TO OS (Added if functonality is wanted in operating system)
//OS_YF 				:= tbYF;
//OS_BB 				:= tbBB;
//OS_BU 				:= tbBU;


// Writing to outputs
Y  						:= tbY;
YF 						:= tbYF;
BB 						:= tbBB;
BU 						:= tbBU;
BX 						:= tbBX;

END_FUNCTION_BLOCK

// Device/Application/MA
FUNCTION_BLOCK MA

// The MA function template shall be used for scaling, display (indication) and monitoring
// (alarming) of process variable or control variable. The template comprises handling of field
// instrument and signaling faults.

VAR_INPUT


	X 		: REAL; // Normal function input
	

	XF 		: BOOL; // External Fault
	

	FBHH 	: BOOL; // Force blocking alarm HH
	
	
	FBLL	: BOOL; // Force blocking alarm LL
	
	
	FUHH	: BOOL; // Force suppression alarm HH
	

	FUWH	: BOOL; // Force suppression alarm WH
	

	FUWL	: BOOL; // Force suppression alarm WL
	
	
	FULL	: BOOL; // Force suppression alarm LL
	
END_VAR

VAR_OUTPUT
	{Analogue output signal FROM FUNCTION template}
	Y		: REAL; // Normal function output
	
	{YF = 1 IF XF = 1 OR IF an INTERNAL error has been detected in the template OR IF an error is detected on the input X.}
	YF		: BOOL; // Function failed
	
	{TRUE, when X*-value >AHH LIMIT. Subjected TO blocking AND suppression.}
	AHH		: BOOL; // Action alarm HH
	
	{Status alarm annunciation (HH) without blocking logic. Subjected TO suppression}
	BHH		: BOOL; // Status alarm HH
	
	{TRUE, when X*-value >WH LIMIT. Subjected TO suppression. Should NOT be used FOR downstream logic.}
	WH		: BOOL; // Warning alarm - WH
	
	{TRUE, when X*-value <WL LIMIT. Subjected TO suppression. Should NOT be used FOR downstream logic.}
	WL		: BOOL; // Warning alarm - WL
	
	
	ALL		: BOOL; // Action alarm LL
	

	BLL		: BOOL; // Status alarm LL
	
	
	BBHH	: BOOL; // Action alarm HH is blocked
	
	
	BBLL	: BOOL; // Action alarm LL is blocked
	

	BU		: BOOL; // Status suppressed
	
	
	BB		: BOOL; // Status blocked
	
	
	BXHH	: BOOL; // Status event HH
	

	BXH		: BOOL; // Status event H
	
	
	BXL		: BOOL; // Status event L
	
	
	BXLL	: BOOL; // Status event LL		
END_VAR

VAR
	srScaledX_Last_Good : REAL;		//Stored scaledX last good measure	
END_VAR

VAR RETAIN
	
	PAHH 	: REAL; 		// Limit AHH
	
	
	PWH		: REAL; 		// Limit WH
	
	
	PWL		: REAL; 		// Limit WL
	
	
	PALL	: REAL; 		// Limit ALL
	
	
	PBXHH	: REAL; 		// Limit BXHH
	
	
	PBXH	: REAL; 		// Limit BXH
	
	
	PBXL	: REAL; 		// Limit BXL
	
	
	PBXLL	: REAL; 		// Limit BXLL
	
	
	PtdA	: TIME := T#0S; // Time delay action alarm 
	
	
	PtdW	: TIME := T#0S; // Time delay warning alarm
	
	
	PHy		: REAL := 0.0; 	// Hysteresis value
	

	PYHR	: REAL; 		// Maximum range
	

	PYLR	: REAL; 		// Minimum range
	

	PEF		: INT := 1;  	// Fault function
	
	Pfbv	: REAL:= 0.0;	// Fall back value
	
	Pdb		: REAL:= 0.0; 	// Dead band
	
END_VAR

VAR
//FunctionBlocks
AHHanalougeAlarm		: fbAnalougeAlarm;		//FB
ALLanalougeAlarm		: fbAnalougeAlarm;		//FB
WHanalougeAlarm			: fbAnalougeAlarm;		//FB
WLanalougeAlarm			: fbAnalougeAlarm;		//FB
BXHHanalougeAlarm		: fbAnalougeAlarm;		//FB 
BXHanalougeAlarm		: fbAnalougeAlarm;		//FB 
BXLLanalougeAlarm		: fbAnalougeAlarm;		//FB 
BXLanalougeAlarm		: fbAnalougeAlarm;		//FB 
Transf					: LIN_TRAFO();			// Linear transformation

// OS Variavles inputs
OS_FBHH					: BOOL;					// OS Force Block High High
OS_FBLL					: BOOL;					// OS Force Block Low Low 
OS_FULL					: BOOL;					// OS force supression low low
OS_FUHH					: BOOL;					// OS force supression high high
OS_FUWH					: BOOL;					// OS force supression warning high
OS_FUWL					: BOOL;					// OS force supression warning low 
OS_FBU					: BOOL;					// OS force supress AHH, ALL, WH, WL, YF


// OS Variavles outputs
OS_AHH					: BOOL;					// OS
OS_ALL					: BOOL;					// OS
OS_YF					: BOOL;					// OS
OS_WH					: BOOL;					// OS
OS_WL					: BOOL;					// OS

END_VAR


VAR_TEMP
	
ScaledX					: REAL;	// Scaled after linear transformation
internal_error 			: BOOL;	// Error in linear transformation
externalFBerror			: BOOL;	// Error from external function blocks

// Temp variables from inputs
trX 		: REAL;		// Scaled X	
tbXF 		: BOOL;		// External fault 
tbFBHH 		: BOOL;		// Force block action high high
tbFBLL		: BOOL;		// Force block action low low
tbFUHH		: BOOL;		// Force supression action high high
tbFUWH		: BOOL;		// Force supression warning high
tbFUWL		: BOOL;		// Force supression warning low
tbFULL		: BOOL;		// Force supression action low low 

// Temp variables from outputs.
trY			: REAL;		// Temp Normal Output
tbYF		: BOOL;		// Temp Output Fault
tbAHH		: BOOL;		// Temp Action High High
tbBHH		: BOOL;		// Temp Blocked High High
tbWH		: BOOL;		// Temp Warning High
tbWL		: BOOL;		// Temp warning low
tbALL		: BOOL;		// Temp Action Low Low
tbBLL		: BOOL;		// Temp Blocked low low
tbBBHH		: BOOL;		// Temp blocked confirmed high high
tbBBLL		: BOOL;		// Temp blocked confirmed low low 
tbBU		: BOOL;		// Temp supressed status
tbBB		: BOOL;		// Temp blocked status
tbBXHH		: BOOL;		// Temp event high high
tbBXH		: BOOL;		// Temp event high
tbBXL		: BOOL;		// Temp event low 
tbBXLL		: BOOL;		// Temp event low low 

END_VAR

VAR CONSTANT
	crXmin 				: REAL 		:= 5530; 
	crXmax : REAL := 32767;
	ciAnalougeHigh 		: SINT 		:= 1;
	ciAnalougeLOW 		: SINT		:= 2;
END_VAR





// Initialising temporary variables
// Handle inputs

trX 		:= X;
tbXF 		:= XF;
tbFBHH 		:= FBHH;
tbFBLL		:= FBLL;
tbFUHH		:= FUHH;
tbFUWH		:= FUWH;
tbFUWL		:= FUWL;
tbFULL		:= FULL;

//Pfbv within range
IF (Pfbv>PYHR) THEN
	Pfbv := PYHR;
ELSIF (Pfbv < PYLR) THEN
	Pfbv := PYLR;	
END_IF

//PEF witin range
IF (PEF<1) THEN
	PEF := 1;
ELSIF (PEF > 3) THEN
	PEF := 1;	
END_IF

//Deadband on X, prescale, 4mA = 5530
IF ((trX >= crXmin-crXmin*((Pdb/100)/2)) AND (trX <= crXmin+crXmin*((Pdb/100)/2))) THEN
	trX := crXmin;
END_IF


Transf(
	IN		:= trX , 
	IN_MIN	:= crXmin, 
	IN_MAX	:= crXmax, 
	OUT_MIN	:= PYLR, 
	OUT_MAX	:= PYHR, 
	OUT		=> ScaledX, 
	ERROR	=> internal_error);






// Handle fault  
IF (tbXF OR internal_error OR externalFBerror) AND NOT (tbFUHH) AND NOT (tbFULL) THEN
	tbYF := TRUE;
	ELSE
	tbYF := FALSE;
END_IF


// ACTION HIGH HIGH 
AHHanalougeAlarm(
	X:=scaledX, 
	PL:= PAHH, 
	PTDH:=PTDA, 
	PTDL:=T#0S , 
	PHY:=PHy, 
	PI:= ciAnalougeHigh , 
	Y=> tbAHH, 
	YF=> externalFBerror, 
	BA=> tbBHH);

// Handle suppression Action High High
IF (tbFUHH OR OS_FUHH) THEN	
    tbBHH := FALSE;
	tbAHH := FALSE;  
END_IF

// Handle output blocked indication Action High High
IF (tbFBHH OR OS_FBHH) THEN
		tbAHH  := FALSE;
		tbBBHH := TRUE;			
ELSE
    tbAHH_Timer := FALSE;
END_IF



// ACTION LOW LOW  
ALLanalougeAlarm(
	X:=scaledX, 
	PL:= PALL, 
	PTDH:=PTDA, 
	PTDL:=T#0S , 
	PHY:=PHy, 
	PI:= ciAnalougeLOW , 
	Y=> tbALL, 
	YF=> externalFBerror, 
	BA=> tbBLL);

// Handle suppression Action Low Low
IF (tbFULL OR OS_FULL) THEN	
    tbBLL := FALSE;
	tbALL := FALSE;  
END_IF

// Handle block Action low low
IF (tbFBLL OR OS_FBLL) THEN
		tbALL  := FALSE;
		tbBBLL := TRUE;			
ELSE
		tbBBLL := FALSE;		
END_IF



// Handle Warning High
WHanalougeAlarm(
	X:= scaledX , 
	PL:= PWH, 
	PTDH:= PTDW, 
	PTDL:= T#0S, 
	PHY:= PHy, 
	PI:= ciAnalougeHigh, 
	Y=> tbWH, 
	YF=> externalFBerror, 
	BA=> );

// Handle suppression warning high
IF (tbFUWH OR OS_FUWH) THEN    
    tbWH := FALSE;
END_IF




// Handle Warning LOW
WLanalougeAlarm(
	X:= scaledX , 
	PL:= PWL, 
	PTDH:= PTDW, 
	PTDL:= T#0S, 
	PHY:= PHy, 
	PI:= ciAnalougeLOW, 
	Y=> tbWL, 
	YF=> externalFBerror, 
	BA=> );


// Handle supression Warning Low
IF (tbFUWL OR OS_FUWL)  THEN
    tbWL := FALSE;
END_IF



// Handle Event High High 
BXHHanalougeAlarm(
	X:= scaledX, 
	PL:= PBXHH, 
	PTDH:= PTDA, 
	PTDL:= T#0S, 
	PHY:= PHy, 
	PI:= ciAnalougeHIGH, 
	Y=> tbBXHH, 
	YF=> externalFBerror, 
	BA=> );



// Handle Event High 
BXHanalougeAlarm(
	X:= scaledX, 
	PL:= PBXH, 
	PTDH:= PTDA, 
	PTDL:= T#0S, 
	PHY:= PHy, 
	PI:= ciAnalougeHIGH, 
	Y=> tbBXH, 
	YF=> externalFBerror, 
	BA=> );


// Handle Event Low Low
BXLLanalougeAlarm(
	X:= scaledX, 
	PL:= PBXLL, 
	PTDH:= PTDA, 
	PTDL:= T#0S, 
	PHY:= PHy, 
	PI:= ciAnalougeLOW, 
	Y=> tbBXLL, 
	YF=> externalFBerror, 
	BA=> );


// Handle Event Low 
BXLanalougeAlarm(
	X:= scaledX, 
	PL:= PBXL, 
	PTDH:= PTDA, 
	PTDL:= T#0S, 
	PHY:= PHy, 
	PI:= ciAnalougeLOW, 
	Y=> tbBXL, 
	YF=> externalFBerror, 
	BA=> );


//Handle blocked binary confirmed
IF (FBHH OR FBLL) THEN	
	tbBB := TRUE;
	ELSE
	tbBB := FALSE;
END_IF


//Handle supressed binary confirmed
IF (FUHH OR FULL OR FUWH OR FUWL) THEN	
	tbBU := TRUE;
	ELSE
	tbBU := FALSE;
END_IF

//Handle OS force supression
IF OS_FBU THEN	
	tbAHH := FALSE;
	tbALL := FALSE;
	tbWH  := FALSE;
	tbWL  := FALSE;
	tbYF  := FALSE;
END_IF


// Handle fault function
IF (tbYF) THEN
	
	CASE PEF OF
	1: trY := srScaledX_Last_Good;						//Freeze last good
		
	2: try := scaledX;									//Show current.
	
	3: trY := Pfbv;										//Substitute value
	
	END_CASE;
ELSE
	
	IF ((scaledX >= PYLR) AND (scaledX <= PYHR)) THEN	//Set last good
			srScaledX_Last_Good := scaledX;
	END_IF;
	trY := scaledX;
END_IF



// Writing to outputs
Y 		:=	trY; 		
YF		:=	tbYF;		
AHH		:=	tbAHH;		
BHH		:=	tbBHH;
WH		:=	tbWH;
WL		:=	tbWL;
ALL		:=	tbALL;
BLL		:=	tbBLL;
BBHH	:=	tbBBHH;
BBLL	:=	tbBBLL;
BU		:=	tbBU;
BB		:=	tbBB;
BXHH	:=	tbBXHH;
BXH		:=	tbBXH;
BXL		:=	tbBXL;
BXLL	:=	tbBXLL;

END_FUNCTION_BLOCK

// Device/Application/fbAnalougeAlarm
FUNCTION_BLOCK fbAnalougeAlarm
VAR_INPUT
	X		 		: REAL; // INPUT
	PL				: REAL; // LIMIT
	PTDH	 		: TIME;	// ONDELAY TIME
	PTDL			: TIME;	// OFFDELAY TIME
	PHY				: REAL;  // Hysteresis
	
END_VAR
VAR_OUTPUT
	Y				: BOOL;
	YF				: BOOL;  
END_VAR
VAR
	
	trX		 		: REAL; // INPUT
	trPL			: REAL; // LIMIT
	ttPTDH	 		: TIME;	// ONDELAY TIME
	ttPTDL			: TIME;	// OFFDELAY TIME
	trPHY			: REAL; // Hysteresis
	tbY				: BOOL; // Output
	tbYf			: BOOL; // Output FAULT
	tbTimerStart	: BOOL;
	
	fbTimer01		: fbTimer(); //Timer
	HysteresisReal1 : HysteresisReal(); 
END_VAR


// UNDERLAG FOR PROGRAMERING AV BLOKK HER.
// 
// // HYSTERESIS ALL
// HYSTERESISALL(IN:=REAL_TO_INT(ScaledX) , HIGH:=REAL_TO_INT(PALL*((PHy / 100)/2)+PALL) , LOW:=REAL_TO_INT(PALL-(PALL*((PHy / 100)/2))) , OUT=> tbALL_Hysteresis );
// 
// // ACTION LOW LOW 
// IF (tbALL_Hysteresis) AND NOT (tbFBLL) AND NOT (tbFULL) THEN    
// 	tbALL_Timer  := TRUE;
// ELSE
//     tbALL_Timer := FALSE;
// END_IF


// HANDKE INPUTS

trX				:= X;
trPL			:= PL;
ttPTDH	 		:= PTDH;
ttPTDL			:= PTDL;
trPHY			:= PHY;




//Hysteresis
//HYSTERESISALL(IN:=REAL_TO_INT(ScaledX) , HIGH:=REAL_TO_INT(PALL*((PHy / 100)/2)+PALL) , LOW:=REAL_TO_INT(PALL-(PALL*((PHy / 100)/2))) , OUT=> tbALL_Hysteresis );


HysteresisReal()

// Handle alarm
IF (trX > PL) THEN	
	tbTimerStart := TRUE;		
	
	ELSE
	tbTimerStart := FALSE;
END_IF

//Send to timer
fbTimer01(X		:=tbTimerStart,
		  PTDH	:=ttPTDH, 
		  PTDL	:=ttPTDL, 
		  Y		=> tbY);

//Set outputs
Y				:=tbY;
YF				:=tbYF;

END_FUNCTION_BLOCK

// Device/Application/SBV
FUNCTION_BLOCK SBV
VAR_INPUT
	XGH            : BOOL;                		 // eXternal Position High
    XGL            : BOOL;                		 // eXternal Position Low
    XH             : BOOL;                		 // eXternal Switch to Position High - in automatic mode
    XL             : BOOL;                		 // eXternal Switch to Position Low - in automatic mode
	XOH            : BOOL;               		 // eXternal Switch to Posistion High - in local/outside mode
	XOL            : BOOL;               		 // eXternal Switch to Posistion Low - in local/outside mode
	XF             : BOOL;                 		 // eXternal Fault 
	LSH            : BOOL;               		 // Lock Safeguard High
	LSL            : BOOL;               		 // Lock Safeguard Low
	FSH            : BOOL;                		 // Force Safeguarding High
    FSL            : BOOL;                		 // [Priority] Force Safeguarding Low
    FDH            : BOOL;              		 // Force Disable High
    FDL            : BOOL;             		     // [Priority] Force Disable Low
	FB             : BOOL;             		     // Force Block	
	FU             : BOOL;						 // Force Supression
	LA             : BOOL;               		 // Set Auto
	LM             : BOOL;               		 // [Priority 2]Set Manual
	LO             : BOOL;               		 // [Priority 1]Set Outside
    //RX             : BOOL;               		 // Reset Fault	
END_VAR

VAR_INPUT RETAIN 								// 
    PFFD           	: TIME := T#5S;       		// Feedback failure delay
    PTDH           	: TIME := T#5S;        	  	// Transit delay low to high
    PTDL           	: TIME := T#5S;       		// Transit delay high to low
    PSTO           	: BOOL;               		// Output YH and YL  constant on.
	PTTO			: TIME := T#2000MS;			// PULS output open YH
	PTTC			: TIME := T#2000MS;			// PULS output close YL
	PAOF			: INT  := 0;				// Parameter action on fault.
	PFT				: INT  := 3;				// Parameter feedback type
	PSUS			: INT  := 0;				// Parameter Template Startup State 
	PSUM			: INT  := 0;				// Parameter for mode at startup
	PSLO			: INT  := 0;				// Parameter for setting local or outside mode
END_VAR

VAR_OUTPUT
	Y              : BOOL;                		// 
	YH             : BOOL;               		// Normal output to switch control element to high state
    YL             : BOOL;                		// Normal output to switch control element to low state
    YF             : BOOL;                		// Control element fault
    BCH            : BOOL;               		// Binary status confirmed high
    BCL            : BOOL;                		// Binary status confirmed low
	BS             : BOOL;                		// Binary status safeguarding
	BB             : BOOL;                		//
	BU             : BOOL;               		//
    BA             : BOOL;               		// Binary status automatic mode
	BO             : BOOL;                		// 
   // BM             : Bool := true;        	// Binary status manual mode    
   // BD             : Bool;                	// Binary status disabled
    YFI            : INT;               		// Fault information
END_VAR

VAR RETAIN
	
	sbBA           		 : BOOL;               	// Binary status automatic mode, RETAINED for prevstate.

END_VAR


VAR
	siState       		 : INT;                 // State of controlled element
    siNextState   		 : INT;                 // Next state of controlled element
	
	sbLA				: BOOL;
	sbLM				: BOOL;
	
	OS_FB				: BOOL;
	OS_FU				: BOOL;
	OS_XLM				: BOOL;
	OS_XHM				: BOOL;
	
	TimerTransLow		: fbTimer;
	TimerTransHigh		: fbTimer;
	TimerFeedbackLow	: fbTimer;
	TimerFeedbackHigh	: fbTimer;
	OutputPulsHigh		: TP;
	OutputPulsLow		: TP;
	
	
	sbYF            : BOOL;
	sbBUpos			: BOOL;
	sbBUneg			: BOOL;
	
	siFBlastvalue	: INT;
END_VAR

VAR_TEMP

	tbHighCommand  		: BOOL;                 // High command
    tbLowCommand   		: BOOL;                 // Low Command
	tbOutsideLocal		: BOOL;					// Interlock of starting object when in local mode
	
	// INPUTS
	tbXGH            : BOOL;                	// eXternal Position High
    tbXGL            : BOOL;                	// eXternal Position Low
    tbXH             : BOOL;                	// eXternal Switch to Position High - in automatic mode
    tbXL             : BOOL;                	// eXternal Switch to Position Low - in automatic mode
	tbXOH            : BOOL;               		//
	tbXOL            : BOOL;               		// 
	tbXF             : BOOL;                 	// 
	tbLSH            : BOOL;               		// 
	tbLSL            : BOOL;               		// 
	tbFSH            : BOOL;                	// Force Safeguarding High
    tbFSL            : BOOL;                	// [Priority] Force Safeguarding Low
    tbFDH            : BOOL;              		// Force Disable High
    tbFDL            : BOOL;             		// [Priority] Force Disable Low
	tbFB             : BOOL;             		// 
	tbFU             : BOOL;					// 
	tbLA             : BOOL;               		// 
	tbLM             : BOOL;               		// 
	tbLO             : BOOL;               		//
	
	
	// OUTPUTS
	tbY             : BOOL;                		// 
	tbYH            : BOOL;               		// Normal output to switch control element to high state
    tbYL            : BOOL;                		// Normal output to switch control element to low state
    // Flytta til statisk minne tbYF            : BOOL;                		// Control element fault
    tbBCH           : BOOL;               		// Binary status confirmed high
    tbBCL           : BOOL;                		// Binary status confirmed low
	tbBS            : BOOL;                		// Binary status safeguarding
	tbBB            : BOOL;                		//
	tbBU            : BOOL;               		//
    // Flytta til statisk minne: tbBA            : BOOL;               	// Binary status automatic mode (
	tbBO            : BOOL;                		//
	tiYFI			:INT;
	
END_VAR

VAR CONSTANT
	ciInitState         : INT := 0;             // [FSM] Initial State of Control Element
    ciLow               : Int := 1;             // [FSM] Control Element in Low state
    ciTransitHigh       : Int := 2;             // [FSM] Control Element in transit to High state
    ciHigh              : Int := 3;             // [FSM] Control Element in High state
    ciTransitLow        : INT := 4;             // [FSM] Control Element in transit to Low state
	
	ciNoFault           : INT := 0;                  // [FAULT] No Fault Indication
    ciFeedbackFaultHigh : Int := 1;             // [FAULT] Feedback Fault
    ciFeedbackFaultLow  : Int := 2;             // [FAULT] Feedback Fault
    ciTransitHighFault  : Int := 3;             // [FAULT] Transit High Fault
    ciTransitLowFault   : INT := 4;             // [FAULT] Transit Low Fault
	ciExternalFault		: INT := 5;				// [FAULT] External fault
	ciConflictFault		: INT := 6;				// [FAULT] Conflict fault (Safeguard and blocking)
	ciSafeguardFault	: INT := 7;				// [FAULT] [Priority] Safeguard fault (No feedback while executing safeguard command)
	
	ciNoAction			: INT := 0;
	ciClose				: INT := 1;
	ciOpen				: INT := 2;
	
	ciNoFeedback		: INT := 0;
	ciHighFeedback		: INT := 1;
	ciLowFeedback		: INT := 2;
	ciFullFeedback		: INT := 3;
	
	ciStartupClosed		: INT := 0;
	ciStartupOpen		: INT := 1;
	ciStartupFeedback	: INT := 2;
	
	ciModeStartupManual		: INT := 0;			//Sets the mode of the block at startup
	ciModeStartupAuto		: INT := 1;			//Sets the mode of the block at startup
	ciModeStartupPrev		: INT := 2;			//Sets the mode of the block at startup
	
	ciModeLocal				: INT := 0;			// Parameter for setting local mode
	ciModeOutside			: INT := 1;			// Parameter for setting outside mode
END_VAR

//INFO, COPYRIGHT MANGOIPA GROUP INC
//SBV function block



//Populate Temporaries and preset outputs

	tbXGH 	:= XGH;
    tbXGL 	:= XGL;    
    tbXH	:= XH;            
    tbXL	:= XL;   
	tbXOH	:= XOH;     
	tbXOL	:= XOL;           
	tbXF	:= XF;            
	tbLSH	:= LSH;           
	tbLSL	:= LSL;           
	tbFSH	:= FSH;           
    tbFSL	:= FSL;            
    tbFDH	:= FDH;            
    tbFDL	:= FDL;            
	tbFB	:= FB;            
	tbFU	:= FU;            
	tbLA	:= LA;              
	tbLM	:= LM;             
	tbLO	:= LO;       

// Timers

TimerTransLow();
TimerTransHigh();
TimerFeedbackLow();
TimerFeedbackHigh();
OutputPulsHigh();
OutputPulsLow();

TimerTransLow.PTDH		:= PTDH;
TimerTransHigh.PTDH 	:= PTDL;
TimerFeedbackLow.PTDH	:= PFFD;
TimerFeedbackHigh.PTDH	:= PFFD;
OutputPulsHigh.PT		:= PTTO;
OutputPulsLow.PT		:= PTTC;

// Handle external faults, subject to supression
IF (tbXF AND NOT tbFU) THEN
	tiYFI := ciExternalFault;
END_IF


// Handle High output puls YH
IF NOT (siState = ciTransitHigh) THEN
	OutputPulsHigh.IN := FALSE;
END_IF

// Handle Low output puls YL
IF NOT (siState = ciTransitLow) THEN
	OutputPulsLow.IN := FALSE;
END_IF

// Handle lock safeguard mode
IF (tbLSL AND NOT tbFB) THEN
	sbBA 			:= FALSE;		// Set mode to manual
ELSIF (tbLSH AND NOT tbFB) THEN
	sbBA 			:= FALSE;		// Set mode to manual
END_IF


//Mode Control
IF tbLM AND NOT sbLM  THEN
    sbBA                        := FALSE;	// Manual mode, BA = 0
ELSIF tbLA AND NOT sbLA THEN
    sbBA                        := TRUE; 	// Auto mode posetive edge,	BA = 1
END_IF;


// Retrigger posetive edge
sbLA := tbLA;
sbLM := tbLM;

// Outside mode / Local mode.
IF tbLO THEN		
	tbBO := TRUE;
	sbBA := FALSE;
	
	CASE PSLO OF
	ciModeLocal				: 
		tbOutsideLocal := TRUE;
		IF tbXGH THEN
			siState := ciHigh;
		ELSIF tbXGL THEN			
			siState := ciLow;
		END_IF
				

	ciModeOutside			: 
	tbOutsideLocal := FALSE;
	//
	END_CASE
ELSE
	tbBO := FALSE;
END_IF	




// Handling safeguarding BS status
IF (tbLSH OR tbLSL OR tbFSH OR tbFSL) THEN
	tbBS := TRUE;
ELSE
	tbBS := FALSE;
END_IF

// Handling blocking BB status
IF (tbFB OR OS_FB) THEN
	tbBB := TRUE;
ELSE
	tbBB := FALSE;
END_IF

//Blocking blocks safeguard and disable transition modes
IF tbBB THEN
	tbLSL := FALSE;
	tbLSH := FALSE;
	tbFSL := FALSE;
	tbFSH := FALSE;
	tbFDH := FALSE;
	tbFDL := FALSE;
END_IF

// Handling supression BU status ON/OFF
IF (tbFU OR OS_FU) THEN
	tbBU  	:= TRUE;	
ELSE
	tbBU 	:= FALSE;
END_IF

// stores PFT before supression sets to "no feedback" on posetive edge
IF tbBU AND NOT sbBUpos THEN
	siFBlastvalue 	:= PFT;
	PFT				:= ciNoFeedback;
END_IF

// sets PFT to last value on negative edge
IF NOT tbBU AND sbBUneg THEN
	PFT 	:= siFBlastValue;
END_IF


// Posetive edge retrigger
sbBUpos := tbBU;

// Negative edge retrigger
sbBUneg := tbBU;


//High and low commands evaluation (AUTO & MANUAL & OUTSIDE & LSL & LSH FDL & FDH
tbLowCommand                  := (tbXL AND sbBA) OR 										// Auto 
								 (OS_XLM AND NOT sbBA AND NOT tbBO) OR 						// Manuell (Triggered by XLM supressed by Auto & Outside mode)
								 (tbBO AND tbXOL AND NOT tbOutsideLocal) OR 				// Outside (Triggered by XOL if in not local outside mode)	
								 (tbLSL AND NOT tbFB) OR									// Lock Safeguard Low subject by blocking
								 (tbFSL AND NOT tbFB);										// Force safeguard Low subject by blocking
												

tbHighCommand                 := (tbXH AND sbBA) OR 										// Auto
								 (OS_XHM AND NOT sbBA AND NOT tbBO AND NOT tbBS) OR 		// Manuell (Triggered by XLM supressed by Auto & Outside mode
								 (tbBO AND tbXOH AND NOT tbOutsideLocal) OR 				// Outside (Triggered by XOL if in not local outside mode)
								 (tbLSH AND NOT tbFB) OR									// Lock Safeguard Low subject by blocking
								 (tbFSH AND NOT tbFB);										// Force safeguard Low subject by blocking
											//FDH

// Handle force disable high command
IF tbFDH AND NOT tbFB THEN
    tbHighCommand             := FALSE;   //If FDH is true then erase high command, prevent transit to high
END_IF;

// Handle force disable low command
IF tbFDL AND NOT tbFB THEN
    tbLowCommand              := FALSE;   //If FDL is true then erase low command, prevent transit to low
END_IF;

// Handle Force safeguard commands
IF tbFSL THEN
    tbHighCommand             := FALSE;
    tbLowCommand              := NOT tbXGL;    //As long as FSL is true and not correct feedback, force transit to low
	
	// I manuell skal den ha Y = 0 (lukka) etter FSL er ute. (Høgkant OS_XLH?)
ELSIF tbFSH THEN
    tbHighCommand             := NOT tbXGH;    //As long as FSH is true and not correct feedback, force transit to high
    tbLowCommand              := FALSE;
	
	// I manuell skal den ha Y = 1 (lukka) etter FSL er ute.
END_IF;

IF (tbBS AND tbBB) THEN
	tiYFI := ciConflictFault;
END_IF

// Handle parameter action on fault
IF sbYF THEN
	CASE PAOF OF 
		ciNoAction:
			// No action on fault
			sbYF := sbYF;		
		ciClose:
			tbLowCommand := TRUE;		
		ciOpen:
			tbHighCommand := TRUE;		
	END_CASE	
END_IF


// Handle parameter feedbacks
CASE PFT OF
	ciNoFeedback:
		tbXGH := (siState = ciHigh) OR (siState = ciTransitHigh);
		tbXGL := (siState = ciLOW) OR (siState = ciTransitlow);
	ciHighFeedback:
		tbXGL := (siState = ciLOW) OR (siState = ciTransitlow);
	ciLowFeedback:
		tbXGH := (siState = ciHigh) OR (siState = ciTransitHigh);
	ciFullFeedback:
		tbXGH := tbXGH;
		tbXGL := tbXGL;
END_CASE;



//Determine next state
IF tbHighCommand THEN
    siNextState              		 := ciHigh;
ELSIF tbLowCommand THEN
    siNextState              		 := ciLow;
End_If;


//Tilstandsmaskin 
CASE siState OF 
	ciInitState:						//Starttilstand, finner riktig tilstand.
	//Init setup før oppstart 
	CASE PSUM OF						//Sets the mode of the block at startup
			ciModeStartupManual		: 
				sbBA := FALSE;							
			ciModeStartupAuto		: 
				sbBA := TRUE;			
			ciModeStartupPrev		: 
				sbBA := sbBA;
	END_CASE
	
	CASE PSUS OF						//Sets the state of the block
		ciStartupClosed		:  
			siState := ciLow;
		ciStartupOpen		:  
			siState := ciHigh;
		ciStartupFeedback	:  	
			IF tbXGH THEN
				siState := ciHigh;
			ELSIF XGL THEN
				siState := ciLow;		
			END_IF
	END_CASE
	

		
		CASE siNextState OF
			ciHigh: siState			 := ciTransitHigh;
			ciLow :	siState 		 := ciTransitLow;		
		END_CASE	
	
	ciLow:
	
	//Feilhandtering om en ikkje har noen tilbakemelding 
	    IF (NOT tbXGL OR tbXGH) THEN
			
		    TimerFeedbackLow.X := TRUE;	
            IF TimerFeedbackLow.Y THEN
                tiYFI           	:= ciFeedbackFaultLow;
            END_IF;
        ELSE
            TimerFeedbackLow.X := FALSE;
        End_If;

        CASE siNextState OF
            ciHigh :                
                siState      		 := ciTransitHigh;
        END_CASE;
		
	ciTransitHigh:
		
		TimerTransHigh.X 			:= TRUE;
		
		OutputPulsHigh.IN 			:= TRUE;
				
		IF tbXGH THEN
			TimerTransHigh.X 		:= FALSE;
			siState           		:= ciHigh;
		END_IF
			

		IF (TimerTransHigh.Y) THEN
			tiYFI	:= ciTransitHighFault;
		END_IF
		
		CASE siNextState OF
            ciLow :                
                siState     		   := ciTransitLow;
        End_Case;
		
	ciHigh:
	
	//Feilhandtering om en ikkje har noen tilbakemelding 
	    IF (NOT tbXGH OR tbXGL) THEN
			
            TimerFeedbackHigh.X := TRUE;	
            IF TimerFeedbackHigh.Y THEN
                tiYFI           	:= ciFeedbackFaultHigh;
            END_IF;
        ELSE
            TimerFeedbackHigh.X 	:= FALSE;
        End_If;
		
        CASE siNextState OF
            ciLow :
                siState       		  := ciTransitLow;
        End_Case;
	
	ciTransitLow:
	
		TimerTransLow.X 			:= TRUE;		
		OutputPulsLow.IN 			:= TRUE;		
	
		IF tbXGL THEN
			TimerTransLow.X 		:= FALSE;
			siState          		:= ciLOW;
		END_IF
		
			IF (TimerTransLow.Y) THEN
				tiYFI	:= ciTransitLowFault;
			END_IF
		
		CASE siNextState OF
            ciHigh :                
                siState      		  := ciTransitHigh;
        End_Case;	

END_CASE


// Safeguard fault
IF (tbBS AND ((tiYFI = ciFeedbackFaultHigh) OR (tiYFI = ciFeedbackFaultLow))) THEN
	tiYFI := ciSafeguardFault;
END_IF;

// FAULT 
sbYF := (tiYFI > ciNoFault);



//Handle supression 
IF tbBU THEN
	sbYF := FALSE;
END_IF


//Write to output //TATT FRA OLAV DIREKTE
Y										:= 	(siState = ciTransitHigh) OR ((siState = ciHigh));
YH                            			:=	OutputPulsHigh.Q OR (PSTO AND (siState = ciTransitHigh)) ;
YL                           			:= 	OutputPulsLow.Q OR (PSTO AND (siState = ciTransitLow)) ;
BA										:= 	sbBA;
BU										:=  tbBU;
YF                           			:= 	(sbYF);
YFI										:=  tiYFI;
BCH                          			:= 	(siState = ciHigh) AND tbXGH AND NOT tbXGL;
BCL                         			:= 	(siState = ciLow) AND tbXGL AND NOT tbXGH;
BS										:=  tbBS;

//Write to HMI

END_FUNCTION_BLOCK

// Device/Application/SBV
FUNCTION_BLOCK SBV
//The SBV function template shall be used for binary (on/off) control of a flow element by 
//means of changing flow of medium (heat or fluid). Typically controlled elements are valves, 
//dampers, etc
VAR_INPUT
	{Signal FROM LIMIT switch high (XGH = 1 is open flow device)}
	XGH		: BOOL; // Position high feedback
	{Signal FROM LIMIT switch low (XGL = 1 is closed flow device)}
	XGL		: BOOL; // Position low feedback
	{FROM process OR logic TO FUNCTION template which set high signal (Y = 1) TO flow device in auto mode.}
	XH		: BOOL; // External set high
	{FROM process OR logic TO FUNCTION template which set high signal (Y = 0) TO flow device in auto mode}
	XL		: BOOL; // External set low
	{Set high signal (positive edge) TO open flow device in outside mode.}
	XOH		: BOOL;	// External outside set high
	{Set low signal (positive edge) TO close flow device in outside mode}
	XOL		: BOOL; // External set low
	{Loop failure-e.g. I/O card broken.}
	XF		: BOOL; // External fault
	{Safeguarding – LSH = 1 overrules operator inputs. Locks the template in manual mode with Y = 1. Input is subject TO blocking. When signal is reset, the template remains in manual mode AND Y = 1.}
	LSH		: BOOL; // Lock safeguarding high
	{Safeguarding – LSL = 1 overrules operator inputs. Locks the template in manual mode with Y = 0. Input is subject TO blocking. When signal is reset, the template remains in manual mode AND Y = 0.}
	LSL		: BOOL; // Lock safeguarding low
	{Safeguarding – Signal overrules operator inputs forces the Y TO 1. When signal goes low, the template will react TO actual terminal status again IF in auto mode. Signal is subject TO blocking.IF in manual mode, the output (Y) remains high after signal returns TO normal}
	FSH		: BOOL; // Force safeguarding high
	{Safeguarding – Signal overrules operator inputs Forces the template Y TO 0). When signal goes low, the template will react TO actual terminal status again IF in auto mode. Signal is subject TO blocking. IF in manual mode, the output (Y) remains low after signal returns TO normal.}
	FSL		: BOOL; // Force safeguarding low
	{Permissive TO open when FDH = 0 AND prevents element FROM being opened when FDH = 1. Signal is subject TO blocking.}
	FDH		: BOOL; // Force disable transition high
	{Permissive TO close when FDL = 0 AND prevents element FROM being closed when FDL = 1. Signal is subject TO blocking.}	
	FDL		: BOOL; // Force disable transition low
	{FB = 1. Safeguarding ACTION LSH, LSL, FSH, FSL AND disable transition FUNCTION FDH, FDL will be blocked.}
	FB		: BOOL; // Force blocking
	{Alarm annunciation is suppressed, YF = 0 AND status XGL, XGH AND XF are neglected as long as FU = 1.}
	FU		: BOOL; // Force supression
	{Locks the template in auto mode. When LA goes low, the template remains in auto mode}
	LA		: BOOL; // Lock auto
	{Locks the template in manual mode. When LM goes low, the template remains in manual mode.}
	LM		: BOOL; // Lock man
	{Locks the template TO outside mode, AND sets the template TO manual mode. When LO goes low, the template remains in manual mode.}
	LO		: BOOL; // Lock outside
END_VAR
VAR_OUTPUT
	{Command TO flow device, Open Y = 1 AND close Y = 0}
	Y		: BOOL; // Normal function output
	{Pulse open command YH = 1 (one pulse)}
	YH		: BOOL; // Pulsed normal function output high
	{Pulse close command YL = 1 (one pulse)}
	YL		: BOOL; // Pulsed normal function output low
	{YF = 1 IF XF = 1 ref. error handling definition}
	YF		: BOOL; // Function failed
	{Output Y compared TO feedback position high LIMIT switch AND validated as TRUE (BCH = 1 IF Y = 1 AND XGH = 1)}
	BCH		: BOOL; // Output position high confirmed
	{Output Y compared TO feedback position low LIMIT switch AND validated as TRUE (BCL = 1 IF Y = 0 AND BCL = 1).}
	BCL		: BOOL; // Output position low confirmed
	{BS = 1 IF ANY safeguarding input is active.}
	BS		: BOOL; // Status safeguarding
	{BB = 1 IF blocking FROM operator station is TRUE OR FB = 1.}
	BB		: BOOL; // Status blocked
	{BU = 1 IF suppressed FROM operator station is TRUE OR FU = 1}
	BU		: BOOL; // Status suppressed
	{BA = 1 when in auto mode}
	BA		: BOOL; // Status auto/man
	{BO = 1 when set outside FROM operator station OR LO = 1}
	BO		: BOOL; // Status outside
END_VAR
VAR
END_VAR

//Mangler operator station in og ut, ingen parametere

END_FUNCTION_BLOCK

// Device/Application/Simulation/fbValveSim
FUNCTION_BLOCK fbValveSim
VAR_INPUT
	X		: BOOL;
END_VAR
VAR_OUTPUT
	BCL		: BOOL;
	BCH		: BOOL;
END_VAR
VAR
	Trans	: fbTimer();
END_VAR
VAR CONSTANT
	PTH		: TIME := T#1S;
	PTL		: TIME := T#1S;
END_VAR


Trans();
Trans.PTDH := PTH;
Trans.PTDL := PTL;

IF (X) THEN
	
	Trans.X := TRUE;
	
	IF(Trans.Y) THEN
		BCH := TRUE;
		BCL := FALSE;
	END_IF

END_IF

IF (NOT X) THEN

	Trans.X := FALSE;

	IF (NOT Trans.Y) THEN
		BCL := TRUE;
		BCH := FALSE;
	END_IF	
END_IF

END_FUNCTION_BLOCK

// Device/Application/SPE
FUNCTION_BLOCK SPE
VAR_INPUT 	
	XGH             : BOOL;                		 // eXternal Position High
    XH              : BOOL;                		 // eXternal Switch to Position High - in automatic mode
    XL              : BOOL;                		 // eXternal Switch to Position Low - in automatic mode
	XOH             : BOOL;               		 // eXternal Switch to Posistion High - in local/outside mode
	XOL             : BOOL;               		 // eXternal Switch to Posistion Low - in local/outside mode
	XF              : BOOL;                 	 // eXternal Fault 
	XE			    : BOOL;						 // eXternal Enabled
	LSH             : BOOL;               		 // Lock Safeguard High
	LSL             : BOOL;               		 // Lock Safeguard Low
	FSH             : BOOL;                		 // Force Safeguarding High
    FSL             : BOOL;                		 // [Priority] Force Safeguarding Low
    FDH             : BOOL;              		 // Force Disable High
    FDL             : BOOL;             		 // [Priority] Force Disable Low
	FB              : BOOL;             		 // Force Block	
	FU              : BOOL;						 // Force Supression
	LA              : BOOL;               		 // Set Auto
	LM              : BOOL;               		 // [Priority 2]Set Manual
	LO              : BOOL;               		 // [Priority 1]Set Outside
   //RX             : BOOL;               		 // Reset Fault	
END_VAR

VAR_INPUT RETAIN 
	PTD			    : TIME := T#2000MS;			 // Parameter Feedback time failure	
	PTFD	        : TIME := T#2000MS;			 // Parameter time before action when loss of feedback
	PTTO			: TIME := T#2000MS;			 // PULS output open YH
	PTTC			: TIME := T#2000MS;			 // PULS output close YL
	PSUM			: INT  := 0;				 // Parameter for Template startup settings
	PSUS			: INT  := 0;				 // Parameter for Operation mode options
	PSLO			: INT  := 1;				 // Parameter for setting Outside mode type 
	PBXF			: BOOL;						 // Parameter for action on external fault
	PBLF			: BOOL;						 // Parameter for Action on loss of run feedback
	PBRE			: BOOL;						 // Parameter for Restart controller options	
END_VAR

VAR_OUTPUT
	Y               : BOOL;                		 // Normal function output.
	YH              : BOOL;               		 // Normal output to switch control element to high state
    YL              : BOOL;                		 // Normal output to switch control element to low state
    YF              : BOOL;                		 // Control element fault
	YFI				: INT;						 // Fault Information
    BCH             : BOOL;               		 // Binary status confirmed high
    BCL             : BOOL;                		 // Binary status confirmed low
    BA              : BOOL;               		 // Binary status automatic mode
	BO              : BOOL;                		 // Binary status outside
	BS              : BOOL;                		 // Binary status safeguarding
	BB              : BOOL;                		 // Binary status blocked
	BU              : BOOL;               		 // Binary status suppressed
	BXH			    : BOOL;						 // Status external set high
	BXL			    : BOOL;						 // Status external set high	
END_VAR

VAR RETAIN
	//VAR RETAIN
END_VAR

VAR
	
	siState       		: INT;                  // State of controlled element
    siNextState   	 	: INT;                  // Next state of controlled element
	sbYF				: BOOL;					// Output fault variable
	sbLA				: BOOL;					// Set auto variable
	sbLM				: BOOL;					// Set manual variable
	
	OutputPulsHigh		: TP;					// TimerPulse lenght YH
	OutputPulsLow		: TP;					// TimerPulse lenght YL
	TimerFeedback		: fbTimer;				// Timer no feedback error
	TimerFeedbackLoss	: fbTimer;				// Timer loss of feedback error
	
//END_VAR

//VAR_TEMP
	//INPUTS
	tbXGH             : BOOL;                		 // eXternal Position High
    tbXH              : BOOL;                		 // eXternal Switch to Position High - in automatic mode
    tbXL              : BOOL;                		 // eXternal Switch to Position Low - in automatic mode
	tbXOH             : BOOL;               		 // eXternal Switch to Posistion High - in local/outside mode
	tbXOL             : BOOL;               		 // eXternal Switch to Posistion Low - in local/outside mode
	tbXF              : BOOL;                 	 	 // eXternal Fault 
	tbXE			  : BOOL;						 // eXternal Enabled
	tbLSH             : BOOL;               		 // Lock Safeguard High
	tbLSL             : BOOL;               		 // Lock Safeguard Low
	tbFSH             : BOOL;                		 // Force Safeguarding High
    tbFSL             : BOOL;                		 // [Priority] Force Safeguarding Low
    tbFDH             : BOOL;              		     // Force Disable High
    tbFDL             : BOOL;             		 	 // [Priority] Force Disable Low
	tbFB              : BOOL;             			 // Force Block	
	tbFU              : BOOL;						 // Force Supression
	tbLA              : BOOL;               		 // Set Auto
	tbLM              : BOOL;               		 // [Priority 2]Set Manual
	tbLO              : BOOL;               		 // [Priority 1]Set Outside
   //tbRX             : BOOL;               		 // Reset Fault
   
   //OUTPUTS
   	tbY               : BOOL;                		 // Output
	tbYH              : BOOL;               		 // Normal output to switch control element to high state
    tbYL              : BOOL;                		 // Normal output to switch control element to low state    
    tbBCH             : BOOL;               		 // Binary status confirmed high
    tbBCL             : BOOL;                		 // Binary status confirmed low
	tbBS              : BOOL;                		 // Binary status safeguarding
	tbBB              : BOOL;                		 // Binary status blocked
	tbBU              : BOOL;               		 // Binary status supressed
	tbBA              : BOOL;               		 // Binary status automatic mode
	tbBO              : BOOL;                		 // Binary status outside
	tiYFI			  : INT;					   	 // FAULT REGISTER
   
    tbLowCommand	  : BOOL;						 // Low Command
	tbHighCommand	  : BOOL;						 // High Command
	
END_VAR

VAR CONSTANT
	//PSUM
	ciManRun			: INT := 0;				 // [PSUM] Manual and run
	ciManStop			: INT := 1;				 // [PSUM] Manual and stop
	ciAsPrevState		: INT := 2;				 // [PSUM] As previous state
	
	//PSUS
	ciOutManAuto		: INT := 0;		 		 // [PSUS] Possible to switch between outside, manual and automatic mode
	ciManAuto			: INT := 1;				 // [PSUS] Possible to switch between manual and automatic mode
	ciManOut  			: INT := 2;				 // [PSUS] Possible to switch between manual and outside mode
	ciLockedMan			: INT := 3;				 // [PSUS] Locked in manual mode
	ciLockedOut	  		: INT := 4;				 //	[PSUS] Locked in outside mode
	
	//PSLO
	ciOutside			: INT := 0;				 // [PSLO] Outside Mode
	ciLocal				: INT := 1;				 // [PSLO] Local Mode

	//TILSTANDSMASKIN
	ciInitState         : INT := 0;             // [FSM] Initial State of Control Element
    ciLow               : INT := 1;             // [FSM] Control Element in Low state / stopped
    ciTransitHigh       : Int := 2;             // [FSM] Control Element in transit to High state
    ciHigh              : INT := 3;             // [FSM] Control Element in High state / running
    ciTransitLow        : INT := 4;             // [FSM] Control Element in transit to Low state

	//FAULT
	ciNoFault           : INT := 0;             // [FAULT] No Fault Indication
    ciFeedbackFaultHigh : Int := 1;             // [FAULT] Feedback Fault
    ciFeedbackFaultLow  : Int := 2;             // [FAULT] Feedback Fault
    ciTransitHighFault  : INT := 3;             // [FAULT] Transit High Fault, missing feedback
    ciTransitLowFault   : INT := 4;             // [FAULT] Transit Low Fault, missing feedback
	ciExternalFault		: INT := 5;				// [FAULT] External fault
	ciConflictFault		: INT := 6;				// [FAULT] Conflict fault (Safeguard and blocking)
	ciSafeguardFault	: INT := 7;				// [FAULT] [Priority] Safeguard fault (No feedback while executing safeguard command)
		
END_VAR

// Designed by MangoIPA TEAM

// The SBE function template shall be used for binary (on/off) control of flow element of medium 
// (electricity, heat or fluid). The controlled element is a unit, e.g. motor, pump, heater, fan etc. 





//Populate Temporaries and preset outputs

tbXGH 								:= XGH;                		    // eXternal Position High
tbXH            					:= XH;                			// eXternal Switch to Position High - in automatic mode
tbXL            					:= XL;                		 	// eXternal Switch to Position Low - in automatic mode
tbXOH            					:= XOH;               		 	// eXternal Switch to Posistion High - in local/outside mode
tbXOL            					:= XOL;               			// eXternal Switch to Posistion Low - in local/outside mode
tbXF            					:= XF;                 	    	// eXternal Fault 
tbXE            					:= XE;						 	// eXternal Enabled
tbLSH            					:= LSH;               			// Lock Safeguard High
tbLSL            					:= LSL;               			// Lock Safeguard Low
tbFSH            					:= FSH;                		 	// Force Safeguarding High
tbFSL            					:= FSL;                			// [Priority] Force Safeguarding Low
tbFDH            					:= FDH;              		    // Force Disable High
tbFDL            					:= FDL;             		    // [Priority] Force Disable Low
tbFB            					:= FB;             		    	// Force Block	
tbFU            					:= FU;							// Force Supression
tbLA            					:= LA;               			// Set Auto
tbLM            					:= LM;        			 		// [Priority 2]Set Manual
tbLO            					:= LO;               								 // [Priority 1]Set Outside
//tbRX              := RX;               							 // Reset Fault	

// Timers
OutputPulsHigh();							 						// TimerPulse lenght YH
OutputPulsLow ();													// TimerPulse lenght YL
TimerFeedback ();								 					// Timer no feedback error
TimerFeedbackLoss();							 					// Timer loss of feedback error


//Timer parameters ( should be behind restart funct or init)
OutputPulsHigh.PT 					:= PTTO;				     	 // TimerPulse lenght YH
OutputPulsLow.PT					:= PTTC;					     // TimerPulse lenght YL
TimerFeedback.PTDH					:= PTD;					     	 // Timer no feedback error
TimerFeedbackLoss.PTDH				:= PTFD;						 // Timer loss of feedback error


// MODE CONTROLL
// Case of PSUS
// Parameter for Operator Mode Options
CASE PSUS OF
	ciOutManAuto:
	//
	ciManAuto:
	//
	ciManOut:
	//
	ciLockedMan:
	//
	ciLockedOut:
	//
END_CASE

//Mode Controll Auto/Man with flank detection posetiv flank!
IF tbLM AND NOT sbLM  THEN											
    tbBA                       			:= FALSE;					// Manual mode, BA = 0
ELSIF tbLA AND NOT sbLA THEN
    tbBA                       			:= TRUE; 	    			// Auto mode posetive edge,	BA = 1
END_IF;
	
sbLM 									:= tbLM;					// Retrigger posetive edge for Mode Control.
sbLA 									:= tbLA;					// Retrigger posetive edge for Mode Control. 

//Mode Controll // Outside/Local
// Mode Controll - Outside/Local mode.
IF tbLO THEN		
	tbBO 								:= TRUE;					// Sets status outside and force off auto-mode
	tbBA 								:= FALSE;
ELSE
	tbBO 								:= FALSE;		
END_IF;

//LOW AND HIGH COMMAND
//High and low commands evaluation (AUTO & MANUAL & OUTSIDE & LSL & LSH FDL & FDH
tbLowCommand                 		    := (tbXH AND tbBA) OR 										// Auto 
								 		   (tbXOH AND NOT tbBA)OR				 					// Manuell
								 		   (tbXOH AND tbBO);							 				// Outside 	
//								 		   (tbLSL AND NOT tbFB) OR									// Lock Safeguard Low subject by blocking
//								 		   (tbFSL AND NOT tbFB);									// Force safeguard Low subject by blocking
												

tbHighCommand                 			:= (tbXL AND tbBA) OR 										// Auto
								           (tbXOL AND NOT tbBA) OR							 		// Manuell 
								           (tbXOL AND tbBO);							 				// Outside
//								           (tbLSH AND NOT tbFB) OR									// Lock Safeguard Low subject by blocking
//								           (tbFSH AND NOT tbFB);									// Force safeguard Low subject by blocking

//Determine next state
IF tbHighCommand THEN
    siNextState              		    := ciHigh;
ELSIF tbLowCommand THEN
    siNextState              		    := ciLow;
End_If;


CASE siState OF
	//INIT STATE
	ciInitState:
		CASE PSUM OF										// Sets the case of PSUM / Parameter for Template startup settings
			ciManRun:
			siNextState := ciHigh;								// Mangler kode for man
			ciManStop:
			siNextState := ciLow;								// Mangler kode for manuell
			ciAsPrevState:		
			//												// Mangler kode for PrevState
		END_CASE
		
		//Case for handling next state
		CASE siNextState OF
		ciHigh: 
			siState						:= ciTransitHigh;
			
		ciLow :	
			siState 		 			:= ciTransitLow;		
	END_CASE	
		
    ciLow               :
	//
	// TRANSIT TO HIGH STATE
    ciTransitHigh : 
	
		OutputPulsHigh.IN				:= TRUE;													// Starts timers for pulse and feedback
		TimerFeedback.X 				:= TRUE;
		IF tbXGH THEN																				// XGH resets timers
			Timerfeedback.X 		    := FALSE;
			siState 					:= ciHigh;
		END_IF
		
		IF (Timerfeedback.Y) THEN																	// Sets FAULT to YFI
			tiYFI						:= ciTransitHighFault;
		END_IF
		
		CASE siNextState OF																			// Changes state 
            ciLow :                
                siState     		    := ciTransitLow;
        End_Case;
		
    ciHigh              : 
	//
    ciTransitLow        : 
	//
	
END_CASE


//Jobber med case, for å få skallet ferdig, så mode og så safeguarding tenker eg, deretter gå igjennom IEC for å micro-kode og teste.
//kos - TRANSIT HIGH DONE.


// FAULT handling
sbYF 									:= (tiYFI > ciNoFault);


//Write to output 
Y										:= 	(siState = ciTransitHigh) OR ((siState = ciHigh));			
YH                            			:=	OutputPulsHigh.Q;
YL                           			:= 	OutputPulsLow.Q;
YF                           			:= 	(sbYF);
YFI										:=  tiYFI;
BCH										:=  (siState = ciHigh);
BCL										:=  (siState = ciLow);
BS										:=  tbBS;
BB										:=  tbBB; 
BU										:=  tbBU;
BA										:=  tbBA; 		
BO										:=  tbBO; 




//Write to HMI

END_FUNCTION_BLOCK

// Device/Application/test_CFC
PROGRAM test_CFC
VAR
	Mtank : MA;
END_VAR

mTank(); // MA

END_PROGRAM

// Device/Application/Test_Blocks/SBV_1
FUNCTION_BLOCK SBV_1
VAR_INPUT
	XGH            : BOOL;                		 // eXternal Position High
    XGL            : BOOL;                		 // eXternal Position Low
    XH             : BOOL;                		 // eXternal Switch to Position High - in automatic mode
    XL             : BOOL;                		 // eXternal Switch to Position Low - in automatic mode
	XOH            : BOOL;               		 // 
	XOL            : BOOL;               		 // 
	XF             : BOOL;                 		 // 
	LSH            : BOOL;               		 // 
	LSL            : BOOL;               		 // 
	FSH            : BOOL;                		 // Force Safeguarding High
    FSL            : BOOL;                		 // [Priority] Force Safeguarding Low
    FDH            : BOOL;              		 // Force Disable High
    FDL            : BOOL;             		     // [Priority] Force Disable Low
	FB             : BOOL;             		     // 
	FU             : BOOL;						 // 
	LA             : BOOL;               		 // 
	LM             : BOOL;               		 // 
	LO             : BOOL;               		 // 
    //RX             : BOOL;               		 // Reset Fault	
END_VAR

VAR_INPUT RETAIN // Disse er hentet fra Olav sin fasit.
    PFFD           	: TIME := T#5S;       		// Feedback failure delay
    PTDH           	: TIME := T#5S;        	  	// Transit delay low to high
    PTDL           	: TIME := T#5S;       		// Transit delay high to low
    PSTO           	: BOOL;               		// Output YH and YL  constant on.
	PTTO			: TIME := T#2000MS;				// PULS output open YH
	PTTC			: TIME := T#2000MS;				// PULS output close YL
END_VAR

VAR_OUTPUT
	Y              : BOOL;                		// 
	YH             : BOOL;               		// Normal output to switch control element to high state
    YL             : BOOL;                		// Normal output to switch control element to low state
    YF             : BOOL;                		// Control element fault
    BCH            : BOOL;               		// Binary status confirmed high
    BCL            : BOOL;                		// Binary status confirmed low
	BS             : BOOL;                		// Binary status safeguarding
	BB             : BOOL;                		//
	BU             : BOOL;               		//
    BA             : BOOL;               		// Binary status automatic mode
	BO             : BOOL;                		// 
   // BM             : Bool := true;        	// Binary status manual mode    
   // BD             : Bool;                	// Binary status disabled
    YFI            : INT;               		// Fault information
END_VAR


VAR
	siState       		 : INT;                 // State of controlled element
    siNextState   		 : INT;                 // Next state of controlled element
	
	sbLA				: BOOL;
	sbLM				: BOOL;
	
	OS_FB				: BOOL;
	OS_FU				: BOOL;
	OS_XLM				: BOOL;
	OS_XHM				: BOOL;
	
	TimerTransLow		: fbTimer;
	TimerTransHigh		: fbTimer;
	TimerFeedbackLow	: fbTimer;
	TimerFeedbackHigh	: fbTimer;
	OutputPulsHigh		: TP;
	OutputPulsLow		: TP;
	
	sbBA            : BOOL;               		// Binary status automatic mode
END_VAR

VAR_TEMP

	tbHighCommand  		: BOOL;                 // High command
    tbLowCommand   		: BOOL;                 // Low Command
	
	// INPUTS
	tbXGH            : BOOL;                	// eXternal Position High
    tbXGL            : BOOL;                	// eXternal Position Low
    tbXH             : BOOL;                	// eXternal Switch to Position High - in automatic mode
    tbXL             : BOOL;                	// eXternal Switch to Position Low - in automatic mode
	tbXOH            : BOOL;               		//
	tbXOL            : BOOL;               		// 
	tbXF             : BOOL;                 	// 
	tbLSH            : BOOL;               		// 
	tbLSL            : BOOL;               		// 
	tbFSH            : BOOL;                	// Force Safeguarding High
    tbFSL            : BOOL;                	// [Priority] Force Safeguarding Low
    tbFDH            : BOOL;              		// Force Disable High
    tbFDL            : BOOL;             		// [Priority] Force Disable Low
	tbFB             : BOOL;             		// 
	tbFU             : BOOL;					// 
	tbLA             : BOOL;               		// 
	tbLM             : BOOL;               		// 
	tbLO             : BOOL;               		//
	
	
	// OUTPUTS
	tbY             : BOOL;                		// 
	tbYH            : BOOL;               		// Normal output to switch control element to high state
    tbYL            : BOOL;                		// Normal output to switch control element to low state
    tbYF            : BOOL;                		// Control element fault
    tbBCH           : BOOL;               		// Binary status confirmed high
    tbBCL           : BOOL;                		// Binary status confirmed low
	tbBS            : BOOL;                		// Binary status safeguarding
	tbBB            : BOOL;                		//
	tbBU            : BOOL;               		//
    // Flytta til statisk minne: tbBA            : BOOL;               	// Binary status automatic mode (
	tbBO            : BOOL;                		//
	tiYFI			:INT;
	
END_VAR

VAR CONSTANT
	ciInitState         : INT := 0;             // [FSM] Initial State of Control Element
    ciLow               : Int := 1;             // [FSM] Control Element in Low state
    ciTransitHigh       : Int := 2;             // [FSM] Control Element in transit to High state
    ciHigh              : Int := 3;             // [FSM] Control Element in High state
    ciTransitLow        : INT := 4;             // [FSM] Control Element in transit to Low state
	
	ciNoFault           : INT;                  // [FAULT] No Fault Indication
    ciFeedbackFaultHigh : Int := 1;             // [FAULT] Feedback Fault
    ciFeedbackFaultLow  : Int := 2;             // [FAULT] Feedback Fault
    ciTransitHighFault  : Int := 3;             // [FAULT] Transit High Fault
    ciTransitLowFault   : Int := 4;             // [FAULT] Transit Low Fault

	
END_VAR

//INFO, COPYRIGHT MANGOIPA GROUP INC
//SBV function block



//Populate Temporaries and preset outputs

	tbXGH 	:= XGH;
    tbXGL 	:= XGL;    
    tbXH	:= XH;            
    tbXL	:= XL;   
	tbXOH	:= XOH;     
	tbXOL	:= XOL;           
	tbXF	:= XF;            
	tbLSH	:= LSH;           
	tbLSL	:= LSL;           
	tbFSH	:= FSH;           
    tbFSL	:= FSL;            
    tbFDH	:= FDH;            
    tbFDL	:= FDL;            
	tbFB	:= FB;            
	tbFU	:= FU;            
	tbLA	:= LA;              
	tbLM	:= LM;             
	tbLO	:= LO;       

// Timers

TimerTransLow();
TimerTransHigh();
TimerFeedbackLow();
TimerFeedbackHigh();
OutputPulsHigh();
OutputPulsLow();

TimerTransLow.PTDH		:= PTDH;
TimerTransHigh.PTDH 	:= PTDL;
TimerFeedbackLow.PTDH	:= PFFD;
TimerFeedbackHigh.PTDH	:= PFFD;
OutputPulsHigh.PT		:= PTTO;
OutputPulsLow.PT		:= PTTC;

// Handle High output puls YH
IF NOT (siState = ciTransitHigh) THEN
	OutputPulsHigh.IN := FALSE;
END_IF

// Handle Low output puls YL
IF NOT (siState = ciTransitLow) THEN
	OutputPulsLow.IN := FALSE;
END_IF

IF (tbLSL) THEN
	sbBA 			:= FALSE;		// IN MANUAL MODE
END_IF

IF (tbLSH) THEN
	sbBA 			:= FALSE;		// IN AUTO MODE
END_IF

//Mode Control
IF tbLM AND NOT sbLM  THEN
    sbBA                        := FALSE;	// Manual mode, BA = 0
ELSIF tbLA AND NOT sbLA THEN
    sbBA                        := TRUE; // Auto mode posetive edge,	BA = 1
END_IF;

// retrigger posetive edge
sbLA := tbLA;
sbLM := tbLM;


// Outside mode
IF tbLO THEN
	tbBO := TRUE;
ELSE
	tbBO := FALSE;
END_IF

// Handling safeguarding BS status
IF (tbLSH OR tbLSL OR tbFSH OR tbFSL) THEN
	tbBS := TRUE;
ELSE
	tbBS := FALSE;
END_IF

// Handling blocking BB status
IF (tbFB OR OS_FB) THEN
	tbBB := TRUE;
ELSE
	tbBB := FALSE;
END_IF

// Handling supression BU status
IF (tbFU OR OS_FU) THEN
	tbBU := TRUE;
ELSE
	tbBU := FALSE;
END_IF

// Hanlding rest of code

//High and low commands evaluation (AUTO & MANUAL & OUTSIDE & (LSL,LSH))
tbLowCommand                  := (tbXL AND sbBA) OR (OS_XLM AND NOT sbBA) OR (tbBO AND tbXOL) OR (tbLSL) OR (tbFDL);
tbHighCommand                 := (tbXH AND sbBA) OR (OS_XHM AND NOT sbBA) OR (tbBO AND tbXOH) OR (tbLSH) OR (tbFDH);


// Handle force disable high command
IF tbFDH THEN
    tbHighCommand             := FALSE;   //If FDH is true then erase high command, prevent transit to high
END_IF;

// Handle force disable low command
IF tbFDL THEN
    tbLowCommand              := FALSE;   //If FDL is true then erase low command, prevent transit to low
END_IF;

// Handle Force safeguard commands
IF tbFSL THEN
    tbHighCommand             := FALSE;
    tbLowCommand              := NOT tbXGL;    //As long as FSL is true and not correct feedback, force transit to low
	
	// I manuell skal den ha Y = 0 (lukka) etter FSL er ute. (Høgkant OS_XLH?)
ELSIF tbFSH THEN
    tbHighCommand             := NOT tbXGH;    //As long as FSH is true and not correct feedback, force transit to high
    tbLowCommand              := FALSE;
	
	// I manuell skal den ha Y = 1 (lukka) etter FSL er ute.
End_If;




//Determine next state
IF tbHighCommand THEN
    siNextState              		 := ciHigh;
ELSIF tbLowCommand THEN
    siNextState              		 := ciLow;
End_If;


//Tilstandsmaskin 
CASE siState OF 
	ciInitState:						//Starttilstand, finner riktig tilstand.
	
		IF tbXGH THEN
			siState := ciHigh;
		ELSIF XGL THEN
			siState := ciLow;		
		END_IF
		
		CASE siNextState OF
			ciHigh: siState			 := ciTransitHigh;
			ciLow :	siState 		 := ciTransitLow;		
		END_CASE	
	
	ciLow:
	
	//Feilhandtering om en ikkje har noen tilbakemelding 
	    IF (NOT tbXGL OR tbXGH) THEN
			
		    TimerFeedbackLow.X := TRUE;	
            IF TimerFeedbackLow.Y THEN
                tiYFI           	:= ciFeedbackFaultLow;
            END_IF;
        ELSE
            TimerFeedbackLow.X := FALSE;
        End_If;

        CASE siNextState OF
            ciHigh :                
                siState      		 := ciTransitHigh;
        END_CASE;
		
	ciTransitHigh:
		
		TimerTransHigh.X 			:= TRUE;
		
		OutputPulsHigh.IN 			:= TRUE;
				
		IF tbXGH THEN
			TimerTransHigh.X 		:= FALSE;
			siState           		:= ciHigh;
		END_IF
			

		IF (TimerTransHigh.Y) THEN
			tiYFI	:= ciTransitHighFault;
		END_IF
		
		CASE siNextState OF
            ciLow :                
                siState     		   := ciTransitLow;
        End_Case;
		
	ciHigh:
	
	//Feilhandtering om en ikkje har noen tilbakemelding 
	    IF (NOT tbXGH OR tbXGL) THEN
			
            TimerFeedbackHigh.X := TRUE;	
            IF TimerFeedbackHigh.Y THEN
                tiYFI           	:= ciFeedbackFaultHigh;
            END_IF;
        ELSE
            TimerFeedbackHigh.X 	:= FALSE;
        End_If;
		
        CASE siNextState OF
            ciLow :
                siState       		  := ciTransitLow;
        End_Case;
	
	ciTransitLow:
	
		TimerTransLow.X 			:= TRUE;
		
		OutputPulsLow.IN 			:= TRUE;		
	
		IF tbXGL THEN
			TimerTransLow.X 		:= FALSE;
			siState          		:= ciLOW;
		END_IF
		
			IF (TimerTransLow.Y) THEN
				tiYFI	:= ciTransitLowFault;
			END_IF
		
		CASE siNextState OF
            ciHigh :                
                siState      		  := ciTransitHigh;
        End_Case;	

END_CASE


//Write to output //TATT FRA OLAV DIREKTE
Y										:= 	(siState = ciTransitHigh) OR ((siState = ciHigh));
YH                            			:=	OutputPulsHigh.Q OR (PSTO AND (siState = ciTransitHigh)) ;
YL                           			:= 	OutputPulsLow.Q OR (PSTO AND (siState = ciTransitLow)) ;
BA										:= 	sbBA;
YF                           			:= 	(tiYFI > ciNoFault);
BCH                          			:= 	(siState = ciHigh) AND tbXGH AND NOT tbXGL;
BCL                         			:= 	(siState = ciLow) AND tbXGL AND NOT tbXGH;

//Write to HMI

END_FUNCTION_BLOCK

// Device/Application/BUGS
FUNCTION_BLOCK BUGS
VAR_INPUT
END_VAR
VAR_OUTPUT
END_VAR
VAR
END_VAR


// Historia om maurtua og dei forferdelege innsekta som plagar hellig PLS kode

// 1 )  Auto feedback på SBV fungerte halveis. (Simulert full feedback)	-Peter
// 2 )
// 3 )
// 4 )
// 5 )
// 6 )
// 7 )
// 8 )
// 9 )
// 10)
// 11)


// Ting som skal må fiksast/gjerast for å få optimal kode,

// 1 )  	Bedre namngiving								- Peter
// 2 )
// 3 )		Feilhantering									- P/R/V
// 3.1) 	Motorvern, pressostatar, osv osv				- P/R/V
// 4 )		HMI?											- P/R/V
// 5 )		Sekvensblokk for slamhantering					- P/R/V
// 6 )
// 7 )		Høgbelastningsmodus								- P/R/V
// 8 )
// 9 )  Spør Tommy om simultanfelling i Aerob/Anoks		- P/R/V
// 10)
// 11)

END_FUNCTION_BLOCK

// Device/Application/fbDigitalAlarm
FUNCTION_BLOCK fbDigitalAlarm
VAR_INPUT
	X		 		: BOOL; // Input
	PTDH	 		: TIME;	// Ondelay Time
	PTDL			: TIME;	// Offdelay Time
	PI				: SINT; // TriggerValue for input 1 = HIGH, 2 = LOW
	
END_VAR

VAR_OUTPUT
	Y				: BOOL; // Output with delay
	YF				: BOOL; // Output fault
	BA				: BOOL; // Output whithout delay
END_VAR

VAR	
	fbTimer01		: fbTimer; 	//Timer
END_VAR

VAR_TEMP	
	trX		 		: BOOL; // Temp Input
	ttPTDH	 		: TIME;	// Temp Ondelay time
	ttPTDL			: TIME;	// Temp Offdelay time
	tbY				: BOOL; // Temp Output
	tbYf			: BOOL; // Temp Output fault
	tbTimerStart	: BOOL; // Temp Starting timer
END_VAR


// Handling Inputs
trX						:= X;
ttPTDH	 				:= PTDH;
ttPTDL					:= PTDL;

// Handling Fault Conditions
IF (PI = 1) THEN
	tbYF 				:= FALSE;
ELSIF (PI = 2) THEN
	tbYF 				:= FALSE;
ELSE
	tbYF 				:= TRUE;
END_IF

// Output with delay, Trigger on High Edge
IF (PI = 1) THEN
	IF trX THEN
	tbTimerStart 		:= TRUE;
	BA 					:= TRUE;			
	ELSE
	tbTimerStart 		:= FALSE;
	BA 					:= FALSE;
	END_IF
END_IF

// Output with delay, Trigger on Low Edgde
IF (PI = 2) THEN
	IF NOT trX THEN	
	tbTimerStart 		:= TRUE;
	BA 					:= TRUE;			
	ELSE
	tbTimerStart 		:= FALSE;
	BA 					:= FALSE;
	END_IF
END_IF

// Send to timer
fbTimer01(X				:=tbTimerStart,
		  PTDH			:=ttPTDH, 
		  PTDL			:=ttPTDL, 
		  Y				=> tbY);

// Handling outputs
Y						:=tbY;
YF						:=tbYF;

END_FUNCTION_BLOCK

// Device/Application/fbPause
FUNCTION_BLOCK fbPause
VAR_INPUT
	Pause: 						 BOOL;	

